# B&R Automation Studio project CleanChemi_SiteManagementSystem (part 9)

```iecst
		// AS Block 125 - ROSTER5_ENABLE
		MasterConfig_LR[IdxSkids_LR].action_enable[124].cyclic := FALSE;// Read data cyclic
		MasterConfig_LR[IdxSkids_LR].action_param[124].p_pv:= ADR(gCMD_LR[IdxSkids_LR].Write_ENABLE_ROSTER5.wENABLE_ROSTER5);// Store data in this variable
		MasterConfig_LR[IdxSkids_LR].action_param[124].quantity := 1;// Number of items to read
		MasterConfig_LR[IdxSkids_LR].action_param[124].unit := 1;// Unit address - ignore if not specified
		MasterConfig_LR[IdxSkids_LR].action_param[124].start_addr := 4560;// Read from this modbus address
		MasterConfig_LR[IdxSkids_LR].action_param[124].timer := 2;// Refresh timer for this item
		MasterConfig_LR[IdxSkids_LR].action_param[124].type := 6;// Function code for this item (2 := read discrete inputs)

		// AS Block 126 - ROSTER6_ENABLE
		MasterConfig_LR[IdxSkids_LR].action_enable[125].cyclic := FALSE;// Read data cyclic
		MasterConfig_LR[IdxSkids_LR].action_param[125].p_pv:= ADR(gCMD_LR[IdxSkids_LR].Write_ENABLE_ROSTER6.wENABLE_ROSTER6);// Store data in this variable
		MasterConfig_LR[IdxSkids_LR].action_param[125].quantity := 1;// Number of items to read
		MasterConfig_LR[IdxSkids_LR].action_param[125].unit := 1;// Unit address - ignore if not specified
		MasterConfig_LR[IdxSkids_LR].action_param[125].start_addr := 4660;// Read from this modbus address
		MasterConfig_LR[IdxSkids_LR].action_param[125].timer := 2;// Refresh timer for this item
		MasterConfig_LR[IdxSkids_LR].action_param[125].type := 6;// Function code for this item (2 := read discrete inputs)

		// AS Block 127 - ROSTER7_ENABLE
		MasterConfig_LR[IdxSkids_LR].action_enable[126].cyclic := FALSE;// Read data cyclic
		MasterConfig_LR[IdxSkids_LR].action_param[126].p_pv:= ADR(gCMD_LR[IdxSkids_LR].Write_ENABLE_ROSTER7.wENABLE_ROSTER7);// Store data in this variable
		MasterConfig_LR[IdxSkids_LR].action_param[126].quantity := 1;// Number of items to read
		MasterConfig_LR[IdxSkids_LR].action_param[126].unit := 1;// Unit address - ignore if not specified
		MasterConfig_LR[IdxSkids_LR].action_param[126].start_addr := 4760;// Read from this modbus address
		MasterConfig_LR[IdxSkids_LR].action_param[126].timer := 2;// Refresh timer for this item
		MasterConfig_LR[IdxSkids_LR].action_param[126].type := 6;// Function code for this item (2 := read discrete inputs)

		// AS Block 128 - ROSTER8_ENABLE
		MasterConfig_LR[IdxSkids_LR].action_enable[127].cyclic := FALSE;// Read data cyclic
		MasterConfig_LR[IdxSkids_LR].action_param[127].p_pv:= ADR(gCMD_LR[IdxSkids_LR].Write_ENABLE_ROSTER8.wENABLE_ROSTER8);// Store data in this variable
		MasterConfig_LR[IdxSkids_LR].action_param[127].quantity := 1;// Number of items to read
		MasterConfig_LR[IdxSkids_LR].action_param[127].unit := 1;// Unit address - ignore if not specified
		MasterConfig_LR[IdxSkids_LR].action_param[127].start_addr := 4860;// Read from this modbus address
		MasterConfig_LR[IdxSkids_LR].action_param[127].timer := 2;// Refresh timer for this item
		MasterConfig_LR[IdxSkids_LR].action_param[127].type := 6;// Function code for this item (2 := read discrete inputs)

		// AS Block 129 - AC_ALARM_ENABLE
		MasterConfig_LR[IdxSkids_LR].action_enable[128].cyclic := FALSE;// Read data cyclic
		MasterConfig_LR[IdxSkids_LR].action_param[128].p_pv:= ADR(gCMD_LR[IdxSkids_LR].Write_AC_ALARM_ENABLE.wAC_ALARM_ENABLE);// Store data in this variable
		MasterConfig_LR[IdxSkids_LR].action_param[128].quantity := 1;// Number of items to read
		MasterConfig_LR[IdxSkids_LR].action_param[128].unit := 1;// Unit address - ignore if not specified
		MasterConfig_LR[IdxSkids_LR].action_param[128].start_addr := gSkid_LR[IdxSkids_LR].AlarmConfig.wAC_ALARM_ENABLE_ADDR;// Read from this modbus address
		MasterConfig_LR[IdxSkids_LR].action_param[128].timer := 2;// Refresh timer for this item
		MasterConfig_LR[IdxSkids_LR].action_param[128].type := 6;// Function code for this item (2 := read discrete inputs)

		// AS Block 130 - AC_TXT_ENABLE
		MasterConfig_LR[IdxSkids_LR].action_enable[129].cyclic := FALSE;// Read data cyclic
		MasterConfig_LR[IdxSkids_LR].action_param[129].p_pv:= ADR(gCMD_LR[IdxSkids_LR].Write_AC_TXT_ENABLE.wAC_TXT_ENABLE);// Store data in this variable
		MasterConfig_LR[IdxSkids_LR].action_param[129].quantity := 1;// Number of items to read
		MasterConfig_LR[IdxSkids_LR].action_param[129].unit := 1;// Unit address - ignore if not specified
		MasterConfig_LR[IdxSkids_LR].action_param[129].start_addr := gSkid_LR[IdxSkids_LR].AlarmConfig.wAC_TXT_ENABLE_ADDR;// Read from this modbus address
		MasterConfig_LR[IdxSkids_LR].action_param[129].timer := 2;// Refresh timer for this item
		MasterConfig_LR[IdxSkids_LR].action_param[129].type := 6;// Function code for this item (2 := read discrete inputs)

		// AS Block 131 - AC_ACTION
		MasterConfig_LR[IdxSkids_LR].action_enable[130].cyclic := FALSE;// Read data cyclic
		MasterConfig_LR[IdxSkids_LR].action_param[130].p_pv:= ADR(gCMD_LR[IdxSkids_LR].Write_AC_ACTION.wAC_ACTION);// Store data in this variable
		MasterConfig_LR[IdxSkids_LR].action_param[130].quantity := 1;// Number of items to read
		MasterConfig_LR[IdxSkids_LR].action_param[130].unit := 1;// Unit address - ignore if not specified
		MasterConfig_LR[IdxSkids_LR].action_param[130].start_addr := gSkid_LR[IdxSkids_LR].AlarmConfig.wAC_ACTION_ADDR;// Read from this modbus address
		MasterConfig_LR[IdxSkids_LR].action_param[130].timer := 2;// Refresh timer for this item
		MasterConfig_LR[IdxSkids_LR].action_param[130].type := 6;// Function code for this item (2 := read discrete inputs)

		// AS Block 132 - AC_DELAY
		MasterConfig_LR[IdxSkids_LR].action_enable[131].cyclic := FALSE;// Read data cyclic
		MasterConfig_LR[IdxSkids_LR].action_param[131].p_pv:= ADR(gCMD_LR[IdxSkids_LR].Write_AC_DELAY.wAC_DELAY);// Store data in this variable
		MasterConfig_LR[IdxSkids_LR].action_param[131].quantity := 1;// Number of items to read
		MasterConfig_LR[IdxSkids_LR].action_param[131].unit := 1;// Unit address - ignore if not specified
		MasterConfig_LR[IdxSkids_LR].action_param[131].start_addr := gSkid_LR[IdxSkids_LR].AlarmConfig.wAC_DELAY_ADDR;// Read from this modbus address
		MasterConfig_LR[IdxSkids_LR].action_param[131].timer := 2;// Refresh timer for this item
		MasterConfig_LR[IdxSkids_LR].action_param[131].type := 6;// Function code for this item (2 := read discrete inputs)

		// AS Block 133 - AC_OFFSET
		MasterConfig_LR[IdxSkids_LR].action_enable[132].cyclic := FALSE;// Read data cyclic
		MasterConfig_LR[IdxSkids_LR].action_param[132].p_pv:= ADR(gCMD_LR[IdxSkids_LR].Write_AC_OFFSET.wAC_OFFSET);// Store data in this variable
		MasterConfig_LR[IdxSkids_LR].action_param[132].quantity := 1;// Number of items to read
		MasterConfig_LR[IdxSkids_LR].action_param[132].unit := 1;// Unit address - ignore if not specified
		MasterConfig_LR[IdxSkids_LR].action_param[132].start_addr := 31000;// Read from this modbus address
		MasterConfig_LR[IdxSkids_LR].action_param[132].timer := 2;// Refresh timer for this item
		MasterConfig_LR[IdxSkids_LR].action_param[132].type := 6;// Function code for this item (2 := read discrete inputs)

		// AS Block 134 - AC_THRESHOLD
		MasterConfig_LR[IdxSkids_LR].action_enable[133].cyclic := FALSE;// Read data cyclic
		MasterConfig_LR[IdxSkids_LR].action_param[133].p_pv:= ADR(gCMD_LR[IdxSkids_LR].Write_AC_THRESHOLD.wAC_THRESHOLD_SWAPPED);// Store data in this variable
		MasterConfig_LR[IdxSkids_LR].action_param[133].quantity := 2;// Number of items to read
		MasterConfig_LR[IdxSkids_LR].action_param[133].unit := 1;// Unit address - ignore if not specified
		MasterConfig_LR[IdxSkids_LR].action_param[133].start_addr := gSkid_LR[IdxSkids_LR].AlarmConfig.wAC_THRESHOLD_ADDR;// Read from this modbus address
		MasterConfig_LR[IdxSkids_LR].action_param[133].timer := 2;// Refresh timer for this item
		MasterConfig_LR[IdxSkids_LR].action_param[133].type := 16;// Function code for this item (2 := read discrete inputs)

		// --------------------------------------------------------------------
		// FOR Modbus Read/Write
		// --------------------------------------------------------------------

		ModbusTcpMaster_LR[IdxSkids_LR].enable := 1;// Start master
		ModbusTcpMaster_LR[IdxSkids_LR].device:= ADR(interface); // Ethernet device string
		ModbusTcpMaster_LR[IdxSkids_LR].p_cfg := ADR(MasterConfig_LR[IdxSkids_LR]); // Pointer to configuration
		ModbusTcpMaster_LR[IdxSkids_LR].p_log := ADR(logger[0,IdxSkids_LR]);// Pointer to logger string array. The logger information will show communication details. Enable for debugging, disable for production to save system resources.
		ModbusTcpMaster_LR[IdxSkids_LR].port:= 510;
		ModbusTcpMaster_LR[IdxSkids_LR].slave_ip_addr := SLAVE_IP_ADDRESSES_LR[IdxSkids_LR]; // Transfer slave device IP address

	END_FOR;

	StartStop := 1;
END_PROGRAM

PROGRAM _CYCLIC
// --------------------------------------------------------------------
// Cyclic FUNCTION call
// --------------------------------------------------------------------
	IF(StartStop) THEN

		FOR IdxSkids_LR := 0 TO MAX_SKIDS_LR DO

			Modbus_CMD_action;
			Modbus_Status_action;
			Alarms_action;

		END_FOR;

	END_IF

END_PROGRAM

PROGRAM _EXIT

	FOR IdxSkids_LR := 0 TO MAX_SKIDS_LR DO
		ModbusTcpMaster_LR[IdxSkids_LR](enable := FALSE);
	END_FOR;

END_PROGRAM
```

#### Status.st
```iecst
ACTION Modbus_Status_action:

	ModbusTcpMaster_LR[IdxSkids_LR]();

	// Heartbeat Connection Monitor
	IF gSkid_LR[IdxSkids_LR].Pmax_General_Variables.HEARTBEAT = gSkid_LR[IdxSkids_LR].Heartbeat.PREVIOUS_HEARTBEAT THEN
		gSkid_LR[IdxSkids_LR].Heartbeat.UNCHANGED_TIMER(IN := TRUE, PT := T#200s);  // Start the timer if value is unchanged for 120 seconds
	ELSE
		gSkid_LR[IdxSkids_LR].Heartbeat.UNCHANGED_TIMER(IN := FALSE);  // Reset the timer if value changes
	END_IF;

	// If the timer reaches 30 seconds, set the systemOffline bit
	IF gSkid_LR[IdxSkids_LR].Heartbeat.UNCHANGED_TIMER.Q THEN
		gSkid_LR[IdxSkids_LR].Heartbeat.SYSTEM_OFFLINE := TRUE;  // System is offline
	ELSE
		gSkid_LR[IdxSkids_LR].Heartbeat.SYSTEM_OFFLINE := FALSE;  // System is still online
	END_IF;

	gSkid_LR[IdxSkids_LR].Heartbeat.MODBUS_RESET(CLK := gSkid_LR[IdxSkids_LR].Heartbeat.SYSTEM_OFFLINE);

	//Reset Modbus buffer on connection timeout
	IF gSkid_LR[IdxSkids_LR].Heartbeat.MODBUS_RESET.Q THEN
		UNIT_ID_Temp := gModbus_LR[IdxSkids_LR].Modbus_PeroxyMAX.Block1_Int[0];
		UNIT_ID_DOSE_Temp := gModbus_LR[IdxSkids_LR].Modbus_Dosing.Block6_Int[0];
		brsmemset(ADR(gModbus_LR[IdxSkids_LR]),0,SIZEOF(gModbus_LR[IdxSkids_LR]));
		gModbus_LR[IdxSkids_LR].Modbus_PeroxyMAX.Block1_Int[0] := UNIT_ID_Temp;
		gModbus_LR[IdxSkids_LR].Modbus_Dosing.Block6_Int[0] := UNIT_ID_DOSE_Temp;
	END_IF;

	// Update previous value for the next cycle
	gSkid_LR[IdxSkids_LR].Heartbeat.PREVIOUS_HEARTBEAT := gSkid_LR[IdxSkids_LR].Pmax_General_Variables.HEARTBEAT;

	// --------------------------------------------------------------------
	// Reset last error information
	// --------------------------------------------------------------------
	IF(reset_error) THEN
		brsmemset(ADR(ModbusTcpMaster_LR[IdxSkids_LR].last_error), 0, 2);
		reset_error := 0;
	END_IF

	// --------------------------------------------------------------------
	// Final Variable Mapping AND Data Conversion - READ
	// --------------------------------------------------------------------

	// AS Block 1 - 6000 DOSING INT
	gSkid_LR[IdxSkids_LR].Pmax_General_Variables.UNIT_ID := gModbus_LR[IdxSkids_LR].Modbus_PeroxyMAX.Block1_Int[0];
	gSkid_LR[IdxSkids_LR].Pmax_General_Variables.USER_ID := gModbus_LR[IdxSkids_LR].Modbus_PeroxyMAX.Block1_Int[2];
	gSkid_LR[IdxSkids_LR].Pmax_General_Variables.USER_ACCESS := gModbus_LR[IdxSkids_LR].Modbus_PeroxyMAX.Block1_Int[4];
	gSkid_LR[IdxSkids_LR].Pmax_General_Variables.PMAX_HOA := gModbus_LR[IdxSkids_LR].Modbus_PeroxyMAX.Block1_Int[6];
	gSkid_LR[IdxSkids_LR].Pmax_General_Variables.PMAX_STATUS := gModbus_LR[IdxSkids_LR].Modbus_PeroxyMAX.Block1_Int[8];
	gSkid_LR[IdxSkids_LR].Pmax_General_Variables.SCREEN_LOCK := INT_TO_BOOL(gModbus_LR[IdxSkids_LR].Modbus_PeroxyMAX.Block1_Int[10]);
	gSkid_LR[IdxSkids_LR].Pmax_General_Variables.HEARTBEAT := gModbus_LR[IdxSkids_LR].Modbus_PeroxyMAX.Block1_Int[12];
	gSkid_LR[IdxSkids_LR].Sensor_Variables.WASTE_LVL := INT_TO_BOOL(gModbus_LR[IdxSkids_LR].Modbus_PeroxyMAX.Block1_Int[14]);

	gSkid_LR[IdxSkids_LR].Pmax_Pump_101.P101_XS := gModbus_LR[IdxSkids_LR].Modbus_PeroxyMAX.Block1_Int[20];
	gSkid_LR[IdxSkids_LR].Sensor_Variables.XV101 := gModbus_LR[IdxSkids_LR].Modbus_PeroxyMAX.Block1_Int[22];
	gSkid_LR[IdxSkids_LR].Sensor_Variables.XV101_ENABLE := gModbus_LR[IdxSkids_LR].Modbus_PeroxyMAX.Block1_Int[24];
	gSkid_LR[IdxSkids_LR].Pmax_Pump_101.P101_AUTOCAL := gModbus_LR[IdxSkids_LR].Modbus_PeroxyMAX.Block1_Int[26];

	gSkid_LR[IdxSkids_LR].Pmax_Pump_102.P102_XS := gModbus_LR[IdxSkids_LR].Modbus_PeroxyMAX.Block1_Int[32];
	gSkid_LR[IdxSkids_LR].Pmax_Pump_102.P102_WARN := gModbus_LR[IdxSkids_LR].Modbus_PeroxyMAX.Block1_Int[34];
	gSkid_LR[IdxSkids_LR].Pmax_Pump_102.P102_ALARM := gModbus_LR[IdxSkids_LR].Modbus_PeroxyMAX.Block1_Int[36];
	gSkid_LR[IdxSkids_LR].Sensor_Variables.XV102 := gModbus_LR[IdxSkids_LR].Modbus_PeroxyMAX.Block1_Int[38];
	gSkid_LR[IdxSkids_LR].Pmax_Pump_102.P102_AUTOCAL := gModbus_LR[IdxSkids_LR].Modbus_PeroxyMAX.Block1_Int[40];
	gSkid_LR[IdxSkids_LR].Pmax_Pump_102.P102_AUTOADAPT := gModbus_LR[IdxSkids_LR].Modbus_PeroxyMAX.Block1_Int[42];
	gSkid_LR[IdxSkids_LR].Pmax_Pump_102.XV102_ENABLE := gModbus_LR[IdxSkids_LR].Modbus_PeroxyMAX.Block1_Int[44];

	gSkid_LR[IdxSkids_LR].Pmax_Pump_103.P103_XS := gModbus_LR[IdxSkids_LR].Modbus_PeroxyMAX.Block1_Int[48];
	gSkid_LR[IdxSkids_LR].Pmax_Pump_103.P103_WARN := gModbus_LR[IdxSkids_LR].Modbus_PeroxyMAX.Block1_Int[50];
	gSkid_LR[IdxSkids_LR].Pmax_Pump_103.P103_ALARM := gModbus_LR[IdxSkids_LR].Modbus_PeroxyMAX.Block1_Int[52];
	gSkid_LR[IdxSkids_LR].Sensor_Variables.XV103 := gModbus_LR[IdxSkids_LR].Modbus_PeroxyMAX.Block1_Int[54];
	gSkid_LR[IdxSkids_LR].Pmax_Pump_103.P103_AUTOCAL := gModbus_LR[IdxSkids_LR].Modbus_PeroxyMAX.Block1_Int[56];
	gSkid_LR[IdxSkids_LR].Pmax_Pump_103.P103_AUTOADAPT := gModbus_LR[IdxSkids_LR].Modbus_PeroxyMAX.Block1_Int[58];

	gSkid_LR[IdxSkids_LR].Pmax_Pump_104.P104_XS := gModbus_LR[IdxSkids_LR].Modbus_PeroxyMAX.Block1_Int[64];
	gSkid_LR[IdxSkids_LR].Pmax_Pump_104.P104_WARN := gModbus_LR[IdxSkids_LR].Modbus_PeroxyMAX.Block1_Int[66];
	gSkid_LR[IdxSkids_LR].Pmax_Pump_104.P104_ALARM := gModbus_LR[IdxSkids_LR].Modbus_PeroxyMAX.Block1_Int[68];
	gSkid_LR[IdxSkids_LR].Sensor_Variables.XV104 := gModbus_LR[IdxSkids_LR].Modbus_PeroxyMAX.Block1_Int[70];
	gSkid_LR[IdxSkids_LR].Pmax_Pump_104.P104_AUTOCAL := gModbus_LR[IdxSkids_LR].Modbus_PeroxyMAX.Block1_Int[72];
	gSkid_LR[IdxSkids_LR].Pmax_Pump_104.P104_AUTOCAL_PV := gModbus_LR[IdxSkids_LR].Modbus_PeroxyMAX.Block1_Int[74];
	gSkid_LR[IdxSkids_LR].Pmax_Pump_104.P104_AUTOADAPT := gModbus_LR[IdxSkids_LR].Modbus_PeroxyMAX.Block1_Int[76];
	gSkid_LR[IdxSkids_LR].Pmax_Pump_104.XV104_ENABLE := gModbus_LR[IdxSkids_LR].Modbus_PeroxyMAX.Block1_Int[78];

	gSkid_LR[IdxSkids_LR].AlarmConfig.AC_ENABLE := gModbus_LR[IdxSkids_LR].Modbus_PeroxyMAX.Block1_Int[118];
	gSkid_LR[IdxSkids_LR].AlarmConfig.AC_ACTION := gModbus_LR[IdxSkids_LR].Modbus_PeroxyMAX.Block1_Int[120];
	gSkid_LR[IdxSkids_LR].AlarmConfig.AC_DELAY := gModbus_LR[IdxSkids_LR].Modbus_PeroxyMAX.Block1_Int[122];
	gSkid_LR[IdxSkids_LR].AlarmConfig.AC_OFFSET := gModbus_LR[IdxSkids_LR].Modbus_PeroxyMAX.Block1_Int[124];

	// AS Block 2 - 6000 DOSING INT - ROSTER
	gSkid_LR[IdxSkids_LR].RosterContact.Contact1_ENABLE := INT_TO_BOOL(gModbus_LR[IdxSkids_LR].Modbus_PeroxyMAX.Block2_Int[0]);
	IDEC_String(ADR(gSkid_LR[IdxSkids_LR].RosterContact.Phone_Read1),ADR(gModbus_LR[IdxSkids_LR].Modbus_PeroxyMAX.Block2_Int[4]),SIZEOF(gSkid_LR[IdxSkids_LR].RosterContact.Phone_Read1),19);

	gSkid_LR[IdxSkids_LR].RosterContact.Contact2_ENABLE := INT_TO_BOOL(gModbus_LR[IdxSkids_LR].Modbus_PeroxyMAX.Block2_Int[24]);
	IDEC_String(ADR(gSkid_LR[IdxSkids_LR].RosterContact.Phone_Read2),ADR(gModbus_LR[IdxSkids_LR].Modbus_PeroxyMAX.Block2_Int[28]),SIZEOF(gSkid_LR[IdxSkids_LR].RosterContact.Phone_Read2),19);

	gSkid_LR[IdxSkids_LR].RosterContact.Contact3_ENABLE := INT_TO_BOOL(gModbus_LR[IdxSkids_LR].Modbus_PeroxyMAX.Block2_Int[48]);
	IDEC_String(ADR(gSkid_LR[IdxSkids_LR].RosterContact.Phone_Read3),ADR(gModbus_LR[IdxSkids_LR].Modbus_PeroxyMAX.Block2_Int[52]),SIZEOF(gSkid_LR[IdxSkids_LR].RosterContact.Phone_Read3),19);

	gSkid_LR[IdxSkids_LR].RosterContact.Contact4_ENABLE := INT_TO_BOOL(gModbus_LR[IdxSkids_LR].Modbus_PeroxyMAX.Block2_Int[72]);
	IDEC_String(ADR(gSkid_LR[IdxSkids_LR].RosterContact.Phone_Read4),ADR(gModbus_LR[IdxSkids_LR].Modbus_PeroxyMAX.Block2_Int[76]),SIZEOF(gSkid_LR[IdxSkids_LR].RosterContact.Phone_Read4),19);

	gSkid_LR[IdxSkids_LR].RosterContact.Contact5_ENABLE := INT_TO_BOOL(gModbus_LR[IdxSkids_LR].Modbus_PeroxyMAX.Block2_Int[96]);
	IDEC_String(ADR(gSkid_LR[IdxSkids_LR].RosterContact.Phone_Read5),ADR(gModbus_LR[IdxSkids_LR].Modbus_PeroxyMAX.Block2_Int[100]),SIZEOF(gSkid_LR[IdxSkids_LR].RosterContact.Phone_Read5),19);

	gSkid_LR[IdxSkids_LR].RosterContact.Contact6_ENABLE := INT_TO_BOOL(gModbus_LR[IdxSkids_LR].Modbus_PeroxyMAX.Block2_Int[120]);
	IDEC_String(ADR(gSkid_LR[IdxSkids_LR].RosterContact.Phone_Read6),ADR(gModbus_LR[IdxSkids_LR].Modbus_PeroxyMAX.Block2_Int[124]),SIZEOF(gSkid_LR[IdxSkids_LR].RosterContact.Phone_Read6),19);

	gSkid_LR[IdxSkids_LR].RosterContact.Contact7_ENABLE := INT_TO_BOOL(gModbus_LR[IdxSkids_LR].Modbus_PeroxyMAX.Block2_Int[144]);
	IDEC_String(ADR(gSkid_LR[IdxSkids_LR].RosterContact.Phone_Read7),ADR(gModbus_LR[IdxSkids_LR].Modbus_PeroxyMAX.Block2_Int[148]),SIZEOF(gSkid_LR[IdxSkids_LR].RosterContact.Phone_Read7),19);

	gSkid_LR[IdxSkids_LR].RosterContact.Contact8_ENABLE := INT_TO_BOOL(gModbus_LR[IdxSkids_LR].Modbus_PeroxyMAX.Block2_Int[168]);
	IDEC_String(ADR(gSkid_LR[IdxSkids_LR].RosterContact.Phone_Read8),ADR(gModbus_LR[IdxSkids_LR].Modbus_PeroxyMAX.Block2_Int[172]),SIZEOF(gSkid_LR[IdxSkids_LR].RosterContact.Phone_Read8),19);

	// AS Block 3 - 6000 DOSING REAL
	gSkid_LR[IdxSkids_LR].ConversionRatios.EFF_1:= IDEC_REAL_Conv(gModbus_LR[IdxSkids_LR].Modbus_PeroxyMAX.Block3_Real[0]);
	gSkid_LR[IdxSkids_LR].ConversionRatios.EFF_2:= IDEC_REAL_Conv(gModbus_LR[IdxSkids_LR].Modbus_PeroxyMAX.Block3_Real[1]);
	gSkid_LR[IdxSkids_LR].ConversionRatios.NAOH_TO_H2O2:= IDEC_REAL_Conv(gModbus_LR[IdxSkids_LR].Modbus_PeroxyMAX.Block3_Real[2]);
	gSkid_LR[IdxSkids_LR].ConversionRatios.TRI_TO_H2O2:= IDEC_REAL_Conv(gModbus_LR[IdxSkids_LR].Modbus_PeroxyMAX.Block3_Real[3]);
	gSkid_LR[IdxSkids_LR].ConversionRatios.NAOH_TO_TRI:= IDEC_REAL_Conv(gModbus_LR[IdxSkids_LR].Modbus_PeroxyMAX.Block3_Real[4]);

	gSkid_LR[IdxSkids_LR].Pmax_General_Variables.PMAX_CONC:= IDEC_REAL_Conv(gModbus_LR[IdxSkids_LR].Modbus_PeroxyMAX.Block3_Real[8]);
	gSkid_LR[IdxSkids_LR].Pmax_General_Variables.PMAX_RATE:= IDEC_REAL_Conv(gModbus_LR[IdxSkids_LR].Modbus_PeroxyMAX.Block3_Real[9]);
	gSkid_LR[IdxSkids_LR].Pmax_General_Variables.PMAX_PV:= IDEC_REAL_Conv(gModbus_LR[IdxSkids_LR].Modbus_PeroxyMAX.Block3_Real[10]);
	gSkid_LR[IdxSkids_LR].Pmax_General_Variables.NAOH_CONC:= IDEC_REAL_Conv(gModbus_LR[IdxSkids_LR].Modbus_PeroxyMAX.Block3_Real[11]);
	gSkid_LR[IdxSkids_LR].Pmax_General_Variables.NAOH_CONC_OD:= IDEC_REAL_Conv(gModbus_LR[IdxSkids_LR].Modbus_PeroxyMAX.Block3_Real[12]);
	gSkid_LR[IdxSkids_LR].Pmax_General_Variables.HP_CONC:= IDEC_REAL_Conv(gModbus_LR[IdxSkids_LR].Modbus_PeroxyMAX.Block3_Real[13]);
	gSkid_LR[IdxSkids_LR].Pmax_General_Variables.HP_CONC_OD:= IDEC_REAL_Conv(gModbus_LR[IdxSkids_LR].Modbus_PeroxyMAX.Block3_Real[14]);

	gSkid_LR[IdxSkids_LR].Pmax_Pump_101.P101_SP:= IDEC_REAL_Conv(gModbus_LR[IdxSkids_LR].Modbus_PeroxyMAX.Block3_Real[21]);
	gSkid_LR[IdxSkids_LR].Pmax_Pump_101.P101_PV:= IDEC_REAL_Conv(gModbus_LR[IdxSkids_LR].Modbus_PeroxyMAX.Block3_Real[22]);
	gSkid_LR[IdxSkids_LR].Pmax_Pump_101.P101_OP:= IDEC_REAL_Conv(gModbus_LR[IdxSkids_LR].Modbus_PeroxyMAX.Block3_Real[23]);
	gSkid_LR[IdxSkids_LR].Pmax_Pump_101.P101_FQ:= IDEC_REAL_Conv(gModbus_LR[IdxSkids_LR].Modbus_PeroxyMAX.Block3_Real[24]);
	gSkid_LR[IdxSkids_LR].Pmax_Pump_101.P101_TI:= IDEC_REAL_Conv(gModbus_LR[IdxSkids_LR].Modbus_PeroxyMAX.Block3_Real[25]);
	gSkid_LR[IdxSkids_LR].Pmax_Pump_101.P101_PI:= IDEC_REAL_Conv(gModbus_LR[IdxSkids_LR].Modbus_PeroxyMAX.Block3_Real[26]);
	gSkid_LR[IdxSkids_LR].Pmax_Pump_101.P101_PFI:= IDEC_REAL_Conv(gModbus_LR[IdxSkids_LR].Modbus_PeroxyMAX.Block3_Real[27]);
	gSkid_LR[IdxSkids_LR].Pmax_Pump_101.P101_LS:= IDEC_REAL_Conv(gModbus_LR[IdxSkids_LR].Modbus_PeroxyMAX.Block3_Real[28]);
	gSkid_LR[IdxSkids_LR].Pmax_Pump_101.P101_GAIN:= IDEC_REAL_Conv(gModbus_LR[IdxSkids_LR].Modbus_PeroxyMAX.Block3_Real[29]);
	gSkid_LR[IdxSkids_LR].Pmax_Pump_101.P101_STEPADJ:= IDEC_REAL_Conv(gModbus_LR[IdxSkids_LR].Modbus_PeroxyMAX.Block3_Real[30]);
	gSkid_LR[IdxSkids_LR].Pmax_Pump_101.P101_TOTALADJ:= IDEC_REAL_Conv(gModbus_LR[IdxSkids_LR].Modbus_PeroxyMAX.Block3_Real[31]);

	gSkid_LR[IdxSkids_LR].Pmax_Pump_101B.P101B_OP:= IDEC_REAL_Conv(gModbus_LR[IdxSkids_LR].Modbus_PeroxyMAX.Block3_Real[35]);
	gSkid_LR[IdxSkids_LR].Pmax_Pump_101B.P101B_PFI:= IDEC_REAL_Conv(gModbus_LR[IdxSkids_LR].Modbus_PeroxyMAX.Block3_Real[36]);
	gSkid_LR[IdxSkids_LR].Pmax_Pump_101B.P101B_SP:= IDEC_REAL_Conv(gModbus_LR[IdxSkids_LR].Modbus_PeroxyMAX.Block3_Real[37]);
	gSkid_LR[IdxSkids_LR].Pmax_Pump_101B.P101B_LS:= IDEC_REAL_Conv(gModbus_LR[IdxSkids_LR].Modbus_PeroxyMAX.Block3_Real[38]);

	gSkid_LR[IdxSkids_LR].Pmax_Pump_102.P102_SP:= IDEC_REAL_Conv(gModbus_LR[IdxSkids_LR].Modbus_PeroxyMAX.Block3_Real[45]);
	gSkid_LR[IdxSkids_LR].Pmax_Pump_102.P102_PV:= IDEC_REAL_Conv(gModbus_LR[IdxSkids_LR].Modbus_PeroxyMAX.Block3_Real[46]);
	gSkid_LR[IdxSkids_LR].Pmax_Pump_102.P102_OP:= IDEC_REAL_Conv(gModbus_LR[IdxSkids_LR].Modbus_PeroxyMAX.Block3_Real[47]);
	gSkid_LR[IdxSkids_LR].Pmax_Pump_102.P102_PFI:= IDEC_REAL_Conv(gModbus_LR[IdxSkids_LR].Modbus_PeroxyMAX.Block3_Real[48]);
	gSkid_LR[IdxSkids_LR].Pmax_Pump_102.P102_FQ:= IDEC_REAL_Conv(gModbus_LR[IdxSkids_LR].Modbus_PeroxyMAX.Block3_Real[49]);
	gSkid_LR[IdxSkids_LR].Pmax_Pump_102.P102_PFQ:= IDEC_REAL_Conv(gModbus_LR[IdxSkids_LR].Modbus_PeroxyMAX.Block3_Real[50]);
	gSkid_LR[IdxSkids_LR].Pmax_Pump_102.P102_PPI:= IDEC_REAL_Conv(gModbus_LR[IdxSkids_LR].Modbus_PeroxyMAX.Block3_Real[51]);
	gSkid_LR[IdxSkids_LR].Pmax_Pump_102.P102_TI:= IDEC_REAL_Conv(gModbus_LR[IdxSkids_LR].Modbus_PeroxyMAX.Block3_Real[52]);
	gSkid_LR[IdxSkids_LR].Pmax_Pump_102.P102_PI:= IDEC_REAL_Conv(gModbus_LR[IdxSkids_LR].Modbus_PeroxyMAX.Block3_Real[53]);
	gSkid_LR[IdxSkids_LR].Pmax_Pump_102.P102_LS:= IDEC_REAL_Conv(gModbus_LR[IdxSkids_LR].Modbus_PeroxyMAX.Block3_Real[54]);
	gSkid_LR[IdxSkids_LR].Pmax_Pump_102.P102_GAIN:= IDEC_REAL_Conv(gModbus_LR[IdxSkids_LR].Modbus_PeroxyMAX.Block3_Real[55]);
	gSkid_LR[IdxSkids_LR].Pmax_Pump_102.P102_STEPADJ:= IDEC_REAL_Conv(gModbus_LR[IdxSkids_LR].Modbus_PeroxyMAX.Block3_Real[56]);
	gSkid_LR[IdxSkids_LR].Pmax_Pump_102.P102_TOTALADJ:= IDEC_REAL_Conv(gModbus_LR[IdxSkids_LR].Modbus_PeroxyMAX.Block3_Real[57]);

	gSkid_LR[IdxSkids_LR].Pmax_Pump_103.P103_SP:= IDEC_REAL_Conv(gModbus_LR[IdxSkids_LR].Modbus_PeroxyMAX.Block3_Real[59]);
	gSkid_LR[IdxSkids_LR].Pmax_Pump_103.P103_PV:= IDEC_REAL_Conv(gModbus_LR[IdxSkids_LR].Modbus_PeroxyMAX.Block3_Real[60]);
	gSkid_LR[IdxSkids_LR].Pmax_Pump_103.P103_OP:= IDEC_REAL_Conv(gModbus_LR[IdxSkids_LR].Modbus_PeroxyMAX.Block3_Real[61]);
	gSkid_LR[IdxSkids_LR].Pmax_Pump_103.P103_PFI:= IDEC_REAL_Conv(gModbus_LR[IdxSkids_LR].Modbus_PeroxyMAX.Block3_Real[62]);

	// AS Block 4 - 6000 DOSING REAL
	gSkid_LR[IdxSkids_LR].Pmax_Pump_103.P103_FQ:= IDEC_REAL_Conv(gModbus_LR[IdxSkids_LR].Modbus_PeroxyMAX.Block4_Real[0]);
	gSkid_LR[IdxSkids_LR].Pmax_Pump_103.P103_PFQ:= IDEC_REAL_Conv(gModbus_LR[IdxSkids_LR].Modbus_PeroxyMAX.Block4_Real[1]);
	gSkid_LR[IdxSkids_LR].Pmax_Pump_103.P103_PPI:= IDEC_REAL_Conv(gModbus_LR[IdxSkids_LR].Modbus_PeroxyMAX.Block4_Real[2]);
	gSkid_LR[IdxSkids_LR].Pmax_Pump_103.P103_TI:= IDEC_REAL_Conv(gModbus_LR[IdxSkids_LR].Modbus_PeroxyMAX.Block4_Real[3]);
	gSkid_LR[IdxSkids_LR].Pmax_Pump_103.P103_PI:= IDEC_REAL_Conv(gModbus_LR[IdxSkids_LR].Modbus_PeroxyMAX.Block4_Real[4]);
	gSkid_LR[IdxSkids_LR].Pmax_Pump_103.P103_LS:= IDEC_REAL_Conv(gModbus_LR[IdxSkids_LR].Modbus_PeroxyMAX.Block4_Real[5]);
	gSkid_LR[IdxSkids_LR].Pmax_Pump_103.P103_GAIN:= IDEC_REAL_Conv(gModbus_LR[IdxSkids_LR].Modbus_PeroxyMAX.Block4_Real[6]);
	gSkid_LR[IdxSkids_LR].Pmax_Pump_103.P103_STEPADJ:= IDEC_REAL_Conv(gModbus_LR[IdxSkids_LR].Modbus_PeroxyMAX.Block4_Real[7]);
	gSkid_LR[IdxSkids_LR].Pmax_Pump_103.P103_TOTALADJ:= IDEC_REAL_Conv(gModbus_LR[IdxSkids_LR].Modbus_PeroxyMAX.Block4_Real[8]);

	gSkid_LR[IdxSkids_LR].Pmax_Pump_104.P104_SP:= IDEC_REAL_Conv(gModbus_LR[IdxSkids_LR].Modbus_PeroxyMAX.Block4_Real[10]);
	gSkid_LR[IdxSkids_LR].Pmax_Pump_104.P104_PV:= IDEC_REAL_Conv(gModbus_LR[IdxSkids_LR].Modbus_PeroxyMAX.Block4_Real[11]);
	gSkid_LR[IdxSkids_LR].Pmax_Pump_104.P104_OP:= IDEC_REAL_Conv(gModbus_LR[IdxSkids_LR].Modbus_PeroxyMAX.Block4_Real[12]);
	gSkid_LR[IdxSkids_LR].Pmax_Pump_104.P104_PFI:= IDEC_REAL_Conv(gModbus_LR[IdxSkids_LR].Modbus_PeroxyMAX.Block4_Real[13]);
	gSkid_LR[IdxSkids_LR].Pmax_Pump_104.P104_FQ:= IDEC_REAL_Conv(gModbus_LR[IdxSkids_LR].Modbus_PeroxyMAX.Block4_Real[14]);
	gSkid_LR[IdxSkids_LR].Pmax_Pump_104.P104_PFQ:= IDEC_REAL_Conv(gModbus_LR[IdxSkids_LR].Modbus_PeroxyMAX.Block4_Real[15]);
	gSkid_LR[IdxSkids_LR].Pmax_Pump_104.P104_PPI:= IDEC_REAL_Conv(gModbus_LR[IdxSkids_LR].Modbus_PeroxyMAX.Block4_Real[16]);
	gSkid_LR[IdxSkids_LR].Pmax_Pump_104.P104_PI:= IDEC_REAL_Conv(gModbus_LR[IdxSkids_LR].Modbus_PeroxyMAX.Block4_Real[18]);
	gSkid_LR[IdxSkids_LR].Pmax_Pump_104.P104_LS:= IDEC_REAL_Conv(gModbus_LR[IdxSkids_LR].Modbus_PeroxyMAX.Block4_Real[19]);
	gSkid_LR[IdxSkids_LR].Pmax_Pump_104.P104_GAIN:= IDEC_REAL_Conv(gModbus_LR[IdxSkids_LR].Modbus_PeroxyMAX.Block4_Real[20]);
	gSkid_LR[IdxSkids_LR].Pmax_Pump_104.P104_STEPADJ:= IDEC_REAL_Conv(gModbus_LR[IdxSkids_LR].Modbus_PeroxyMAX.Block4_Real[21]);
	gSkid_LR[IdxSkids_LR].Pmax_Pump_104.P104_TOTALADJ:= IDEC_REAL_Conv(gModbus_LR[IdxSkids_LR].Modbus_PeroxyMAX.Block4_Real[22]);

	gSkid_LR[IdxSkids_LR].Sensor_Variables.CD101:= IDEC_REAL_Conv(gModbus_LR[IdxSkids_LR].Modbus_PeroxyMAX.Block4_Real[24]);
	gSkid_LR[IdxSkids_LR].Sensor_Variables.CD101_SP:= IDEC_REAL_Conv(gModbus_LR[IdxSkids_LR].Modbus_PeroxyMAX.Block4_Real[25]);
	gSkid_LR[IdxSkids_LR].Sensor_Variables.CD102:= IDEC_REAL_Conv(gModbus_LR[IdxSkids_LR].Modbus_PeroxyMAX.Block4_Real[26]);
	gSkid_LR[IdxSkids_LR].Sensor_Variables.CD102_SP:= IDEC_REAL_Conv(gModbus_LR[IdxSkids_LR].Modbus_PeroxyMAX.Block4_Real[27]);
	gSkid_LR[IdxSkids_LR].Sensor_Variables.CD103:= IDEC_REAL_Conv(gModbus_LR[IdxSkids_LR].Modbus_PeroxyMAX.Block4_Real[28]);
	gSkid_LR[IdxSkids_LR].Sensor_Variables.CD103_SP:= IDEC_REAL_Conv(gModbus_LR[IdxSkids_LR].Modbus_PeroxyMAX.Block4_Real[29]);

	gSkid_LR[IdxSkids_LR].Sensor_Variables.CD101_TI:= IDEC_REAL_Conv(gModbus_LR[IdxSkids_LR].Modbus_PeroxyMAX.Block4_Real[36]);
	gSkid_LR[IdxSkids_LR].Sensor_Variables.CD102_TI:= IDEC_REAL_Conv(gModbus_LR[IdxSkids_LR].Modbus_PeroxyMAX.Block4_Real[37]);
	gSkid_LR[IdxSkids_LR].Sensor_Variables.CD103_TI:= IDEC_REAL_Conv(gModbus_LR[IdxSkids_LR].Modbus_PeroxyMAX.Block4_Real[38]);

	gSkid_LR[IdxSkids_LR].AlarmConfig.AC_THRESHOLD :=  IDEC_REAL_Conv(gModbus_LR[IdxSkids_LR].Modbus_PeroxyMAX.Block4_Real[44]);
	gSkid_LR[IdxSkids_LR].Pmax_General_Variables.HMI_REV_A:= IDEC_REAL_Conv(gModbus_LR[IdxSkids_LR].Modbus_PeroxyMAX.Block4_Real[45]);
	gSkid_LR[IdxSkids_LR].Pmax_General_Variables.HMI_REV_B:= IDEC_REAL_Conv(gModbus_LR[IdxSkids_LR].Modbus_PeroxyMAX.Block4_Real[46]);
	gSkid_LR[IdxSkids_LR].Pmax_General_Variables.PLC_REV_A:= IDEC_REAL_Conv(gModbus_LR[IdxSkids_LR].Modbus_PeroxyMAX.Block4_Real[47]);
	gSkid_LR[IdxSkids_LR].Pmax_General_Variables.PLC_REV_B:= IDEC_REAL_Conv(gModbus_LR[IdxSkids_LR].Modbus_PeroxyMAX.Block4_Real[48]);

	gSkid_LR[IdxSkids_LR].BufferTank.BT_PERCENT:= IDEC_REAL_Conv(gModbus_LR[IdxSkids_LR].Modbus_PeroxyMAX.Block4_Real[50]);
	gSkid_LR[IdxSkids_LR].BufferTank.LI200:= IDEC_REAL_Conv(gModbus_LR[IdxSkids_LR].Modbus_PeroxyMAX.Block4_Real[51]);
	gSkid_LR[IdxSkids_LR].BufferTank.LSHH200:= IDEC_REAL_Conv(gModbus_LR[IdxSkids_LR].Modbus_PeroxyMAX.Block4_Real[52]);
	gSkid_LR[IdxSkids_LR].BufferTank.DRAINTIME_SP:= IDEC_REAL_Conv(gModbus_LR[IdxSkids_LR].Modbus_PeroxyMAX.Block4_Real[53]);
	gSkid_LR[IdxSkids_LR].BufferTank.DRAINTIME_PV:= IDEC_REAL_Conv(gModbus_LR[IdxSkids_LR].Modbus_PeroxyMAX.Block4_Real[54]);
	gSkid_LR[IdxSkids_LR].BufferTank.FILLTIME_SP:= IDEC_REAL_Conv(gModbus_LR[IdxSkids_LR].Modbus_PeroxyMAX.Block4_Real[55]);
	gSkid_LR[IdxSkids_LR].BufferTank.FILLTIME_PV:= IDEC_REAL_Conv(gModbus_LR[IdxSkids_LR].Modbus_PeroxyMAX.Block4_Real[56]);

	// AS Block 5 - 6000 DOSING REAL - SPARE
	//:= IDEC_REAL_Conv(gModbus_LR[IdxSkids_LR].Modbus_PeroxyMAX.Block5_Real[0]);

	// AS Block 6 - 7000 DOSING INT
	gSkid_LR[IdxSkids_LR].Pmax_General_Variables.UNIT_ID_DOSE := gModbus_LR[IdxSkids_LR].Modbus_Dosing.Block6_Int[0];

	gSkid_LR[IdxSkids_LR].Dosing_Pump_201.P201_XS := gModbus_LR[IdxSkids_LR].Modbus_Dosing.Block6_Int[6];
	gSkid_LR[IdxSkids_LR].Dosing_Pump_201.P201_HOA := gModbus_LR[IdxSkids_LR].Modbus_Dosing.Block6_Int[8];
	gSkid_LR[IdxSkids_LR].Dosing_Pump_201.P201_CHEM := gModbus_LR[IdxSkids_LR].Modbus_Dosing.Block6_Int[10];
	gSkid_LR[IdxSkids_LR].Dosing_Pump_201.P201_ENABLE := gModbus_LR[IdxSkids_LR].Modbus_Dosing.Block6_Int[12];
	gSkid_LR[IdxSkids_LR].Dosing_Pump_201.P201_ADJ := gModbus_LR[IdxSkids_LR].Modbus_Dosing.Block6_Int[14];
	gSkid_LR[IdxSkids_LR].Dosing_Pump_201.P201_PTYPE := gModbus_LR[IdxSkids_LR].Modbus_Dosing.Block6_Int[16];
	gSkid_LR[IdxSkids_LR].Dosing_Pump_201.P201_WARN := gModbus_LR[IdxSkids_LR].Modbus_Dosing.Block6_Int[18];
	gSkid_LR[IdxSkids_LR].Dosing_Pump_201.P201_ALARM := gModbus_LR[IdxSkids_LR].Modbus_Dosing.Block6_Int[20];
	gSkid_LR[IdxSkids_LR].Sensor_Variables.XV201 := gModbus_LR[IdxSkids_LR].Modbus_Dosing.Block6_Int[22];
	gSkid_LR[IdxSkids_LR].Dosing_Pump_201.P201_AUTOCAL := gModbus_LR[IdxSkids_LR].Modbus_Dosing.Block6_Int[24];
	gSkid_LR[IdxSkids_LR].Dosing_Pump_201.P201_AUTOCAL_PV := gModbus_LR[IdxSkids_LR].Modbus_Dosing.Block6_Int[26];
	gSkid_LR[IdxSkids_LR].Dosing_Pump_201.P201_AUTOADAPT := gModbus_LR[IdxSkids_LR].Modbus_Dosing.Block6_Int[28];

	gSkid_LR[IdxSkids_LR].Dosing_Pump_202.P202_XS := gModbus_LR[IdxSkids_LR].Modbus_Dosing.Block6_Int[32];
	gSkid_LR[IdxSkids_LR].Dosing_Pump_202.P202_HOA := gModbus_LR[IdxSkids_LR].Modbus_Dosing.Block6_Int[34];
	gSkid_LR[IdxSkids_LR].Dosing_Pump_202.P202_CHEM := gModbus_LR[IdxSkids_LR].Modbus_Dosing.Block6_Int[36];
	gSkid_LR[IdxSkids_LR].Dosing_Pump_202.P202_ENABLE := gModbus_LR[IdxSkids_LR].Modbus_Dosing.Block6_Int[38];
	gSkid_LR[IdxSkids_LR].Dosing_Pump_202.P202_ADJ := gModbus_LR[IdxSkids_LR].Modbus_Dosing.Block6_Int[40];
	gSkid_LR[IdxSkids_LR].Dosing_Pump_202.P202_WARN := gModbus_LR[IdxSkids_LR].Modbus_Dosing.Block6_Int[42];
	gSkid_LR[IdxSkids_LR].Dosing_Pump_202.P202_ALARM := gModbus_LR[IdxSkids_LR].Modbus_Dosing.Block6_Int[44];
	gSkid_LR[IdxSkids_LR].Sensor_Variables.XV202 := gModbus_LR[IdxSkids_LR].Modbus_Dosing.Block6_Int[46];
	gSkid_LR[IdxSkids_LR].Dosing_Pump_202.P202_AUTOCAL := gModbus_LR[IdxSkids_LR].Modbus_Dosing.Block6_Int[48];
	gSkid_LR[IdxSkids_LR].Dosing_Pump_202.P202_AUTOCAL_PV := gModbus_LR[IdxSkids_LR].Modbus_Dosing.Block6_Int[50];
	gSkid_LR[IdxSkids_LR].Dosing_Pump_202.P202_AUTOADAPT := gModbus_LR[IdxSkids_LR].Modbus_Dosing.Block6_Int[52];

	gSkid_LR[IdxSkids_LR].Dosing_Pump_203.P203_XS := gModbus_LR[IdxSkids_LR].Modbus_Dosing.Block6_Int[56];
	gSkid_LR[IdxSkids_LR].Dosing_Pump_203.P203_HOA := gModbus_LR[IdxSkids_LR].Modbus_Dosing.Block6_Int[58];
	gSkid_LR[IdxSkids_LR].Dosing_Pump_203.P203_CHEM := gModbus_LR[IdxSkids_LR].Modbus_Dosing.Block6_Int[60];
	gSkid_LR[IdxSkids_LR].Dosing_Pump_203.P203_ENABLE := gModbus_LR[IdxSkids_LR].Modbus_Dosing.Block6_Int[62];
	gSkid_LR[IdxSkids_LR].Dosing_Pump_203.P203_ADJ := gModbus_LR[IdxSkids_LR].Modbus_Dosing.Block6_Int[64];
	gSkid_LR[IdxSkids_LR].Dosing_Pump_203.P203_WARN := gModbus_LR[IdxSkids_LR].Modbus_Dosing.Block6_Int[66];
	gSkid_LR[IdxSkids_LR].Dosing_Pump_203.P203_ALARM := gModbus_LR[IdxSkids_LR].Modbus_Dosing.Block6_Int[68];
	gSkid_LR[IdxSkids_LR].Sensor_Variables.XV203 := gModbus_LR[IdxSkids_LR].Modbus_Dosing.Block6_Int[70];
	gSkid_LR[IdxSkids_LR].Dosing_Pump_203.P203_AUTOCAL := gModbus_LR[IdxSkids_LR].Modbus_Dosing.Block6_Int[72];
	gSkid_LR[IdxSkids_LR].Dosing_Pump_203.P203_AUTOCAL_PV := gModbus_LR[IdxSkids_LR].Modbus_Dosing.Block6_Int[74];
	gSkid_LR[IdxSkids_LR].Dosing_Pump_203.P203_AUTOADAPT := gModbus_LR[IdxSkids_LR].Modbus_Dosing.Block6_Int[76];

	// AS Block 7 - 7000 DOSING INT
	gSkid_LR[IdxSkids_LR].Sensor_Variables.SERNSORS_CONFIG := gModbus_LR[IdxSkids_LR].Modbus_Dosing.Block7_Int[104];

	gSkid_LR[IdxSkids_LR].Sensor_Variables.FI301_MODE := gModbus_LR[IdxSkids_LR].Modbus_Dosing.Block7_Int[118];
	gSkid_LR[IdxSkids_LR].Sensor_Variables.FI302_MODE := gModbus_LR[IdxSkids_LR].Modbus_Dosing.Block7_Int[120];
	gSkid_LR[IdxSkids_LR].Sensor_Variables.FI303_MODE := gModbus_LR[IdxSkids_LR].Modbus_Dosing.Block7_Int[122];
	gSkid_LR[IdxSkids_LR].Sensor_Variables.FI304_MODE := gModbus_LR[IdxSkids_LR].Modbus_Dosing.Block7_Int[124];

	// AS Block 8 - 7000 DOSING REAL
	gSkid_LR[IdxSkids_LR].Dosing_Pump_201.P201_REF_SENSOR := IDEC_REAL_Conv(gModbus_LR[IdxSkids_LR].Modbus_Dosing.Block8_Real[0]);
	gSkid_LR[IdxSkids_LR].Dosing_Pump_201.P201_CONC := IDEC_REAL_Conv(gModbus_LR[IdxSkids_LR].Modbus_Dosing.Block8_Real[1]);
	gSkid_LR[IdxSkids_LR].Dosing_Pump_201.P201_PPM := IDEC_REAL_Conv(gModbus_LR[IdxSkids_LR].Modbus_Dosing.Block8_Real[2]);
	gSkid_LR[IdxSkids_LR].Dosing_Pump_201.P201_APPM := IDEC_REAL_Conv(gModbus_LR[IdxSkids_LR].Modbus_Dosing.Block8_Real[3]);
	gSkid_LR[IdxSkids_LR].Dosing_Pump_201.P201_SP := IDEC_REAL_Conv(gModbus_LR[IdxSkids_LR].Modbus_Dosing.Block8_Real[4]);
	gSkid_LR[IdxSkids_LR].Dosing_Pump_201.P201_PV := IDEC_REAL_Conv(gModbus_LR[IdxSkids_LR].Modbus_Dosing.Block8_Real[5]);
	gSkid_LR[IdxSkids_LR].Dosing_Pump_201.P201_OP := IDEC_REAL_Conv(gModbus_LR[IdxSkids_LR].Modbus_Dosing.Block8_Real[6]);
	gSkid_LR[IdxSkids_LR].Dosing_Pump_201.P201_PFI := IDEC_REAL_Conv(gModbus_LR[IdxSkids_LR].Modbus_Dosing.Block8_Real[7]);
	gSkid_LR[IdxSkids_LR].Dosing_Pump_201.P201_FQ := IDEC_REAL_Conv(gModbus_LR[IdxSkids_LR].Modbus_Dosing.Block8_Real[8]);
	gSkid_LR[IdxSkids_LR].Dosing_Pump_201.P201_PI := IDEC_REAL_Conv(gModbus_LR[IdxSkids_LR].Modbus_Dosing.Block8_Real[9]);
	gSkid_LR[IdxSkids_LR].Dosing_Pump_201.P201_TI := IDEC_REAL_Conv(gModbus_LR[IdxSkids_LR].Modbus_Dosing.Block8_Real[10]);
	gSkid_LR[IdxSkids_LR].Dosing_Pump_201.P201_PFQ := IDEC_REAL_Conv(gModbus_LR[IdxSkids_LR].Modbus_Dosing.Block8_Real[11]);
	gSkid_LR[IdxSkids_LR].Dosing_Pump_201.P201_PPI := IDEC_REAL_Conv(gModbus_LR[IdxSkids_LR].Modbus_Dosing.Block8_Real[12]);
	gSkid_LR[IdxSkids_LR].Dosing_Pump_201.P201_LS := IDEC_REAL_Conv(gModbus_LR[IdxSkids_LR].Modbus_Dosing.Block8_Real[13]);
	gSkid_LR[IdxSkids_LR].Dosing_Pump_201.P201_ASP := IDEC_REAL_Conv(gModbus_LR[IdxSkids_LR].Modbus_Dosing.Block8_Real[14]);
	gSkid_LR[IdxSkids_LR].Dosing_Pump_201.P201_GAIN := IDEC_REAL_Conv(gModbus_LR[IdxSkids_LR].Modbus_Dosing.Block8_Real[15]);
	gSkid_LR[IdxSkids_LR].Dosing_Pump_201.P201_STEPADJ := IDEC_REAL_Conv(gModbus_LR[IdxSkids_LR].Modbus_Dosing.Block8_Real[16]);
	gSkid_LR[IdxSkids_LR].Dosing_Pump_201.P201_TOTALADJ := IDEC_REAL_Conv(gModbus_LR[IdxSkids_LR].Modbus_Dosing.Block8_Real[17]);

	gSkid_LR[IdxSkids_LR].Dosing_Pump_202.P202_REF_SENSOR := IDEC_REAL_Conv(gModbus_LR[IdxSkids_LR].Modbus_Dosing.Block8_Real[19]);
	gSkid_LR[IdxSkids_LR].Dosing_Pump_202.P202_CONC := IDEC_REAL_Conv(gModbus_LR[IdxSkids_LR].Modbus_Dosing.Block8_Real[20]);
	gSkid_LR[IdxSkids_LR].Dosing_Pump_202.P202_PPM := IDEC_REAL_Conv(gModbus_LR[IdxSkids_LR].Modbus_Dosing.Block8_Real[21]);
	gSkid_LR[IdxSkids_LR].Dosing_Pump_202.P202_APPM := IDEC_REAL_Conv(gModbus_LR[IdxSkids_LR].Modbus_Dosing.Block8_Real[22]);
	gSkid_LR[IdxSkids_LR].Dosing_Pump_202.P202_SP := IDEC_REAL_Conv(gModbus_LR[IdxSkids_LR].Modbus_Dosing.Block8_Real[23]);
	gSkid_LR[IdxSkids_LR].Dosing_Pump_202.P202_PV := IDEC_REAL_Conv(gModbus_LR[IdxSkids_LR].Modbus_Dosing.Block8_Real[24]);
	gSkid_LR[IdxSkids_LR].Dosing_Pump_202.P202_OP := IDEC_REAL_Conv(gModbus_LR[IdxSkids_LR].Modbus_Dosing.Block8_Real[25]);
	gSkid_LR[IdxSkids_LR].Dosing_Pump_202.P202_PFI := IDEC_REAL_Conv(gModbus_LR[IdxSkids_LR].Modbus_Dosing.Block8_Real[26]);
	gSkid_LR[IdxSkids_LR].Dosing_Pump_202.P202_FQ := IDEC_REAL_Conv(gModbus_LR[IdxSkids_LR].Modbus_Dosing.Block8_Real[27]);
	gSkid_LR[IdxSkids_LR].Dosing_Pump_202.P202_PI := IDEC_REAL_Conv(gModbus_LR[IdxSkids_LR].Modbus_Dosing.Block8_Real[28]);
	gSkid_LR[IdxSkids_LR].Dosing_Pump_202.P202_TI := IDEC_REAL_Conv(gModbus_LR[IdxSkids_LR].Modbus_Dosing.Block8_Real[29]);
	gSkid_LR[IdxSkids_LR].Dosing_Pump_202.P202_PFQ := IDEC_REAL_Conv(gModbus_LR[IdxSkids_LR].Modbus_Dosing.Block8_Real[30]);
	gSkid_LR[IdxSkids_LR].Dosing_Pump_202.P202_PPI := IDEC_REAL_Conv(gModbus_LR[IdxSkids_LR].Modbus_Dosing.Block8_Real[31]);
	gSkid_LR[IdxSkids_LR].Dosing_Pump_202.P202_LS := IDEC_REAL_Conv(gModbus_LR[IdxSkids_LR].Modbus_Dosing.Block8_Real[32]);
	gSkid_LR[IdxSkids_LR].Dosing_Pump_202.P202_ASP := IDEC_REAL_Conv(gModbus_LR[IdxSkids_LR].Modbus_Dosing.Block8_Real[33]);
	gSkid_LR[IdxSkids_LR].Dosing_Pump_202.P202_GAIN := IDEC_REAL_Conv(gModbus_LR[IdxSkids_LR].Modbus_Dosing.Block8_Real[34]);
	gSkid_LR[IdxSkids_LR].Dosing_Pump_202.P202_STEPADJ := IDEC_REAL_Conv(gModbus_LR[IdxSkids_LR].Modbus_Dosing.Block8_Real[35]);
	gSkid_LR[IdxSkids_LR].Dosing_Pump_202.P202_TOTALADJ := IDEC_REAL_Conv(gModbus_LR[IdxSkids_LR].Modbus_Dosing.Block8_Real[36]);

	gSkid_LR[IdxSkids_LR].Dosing_Pump_203.P203_REF_SENSOR := IDEC_REAL_Conv(gModbus_LR[IdxSkids_LR].Modbus_Dosing.Block8_Real[38]);
	gSkid_LR[IdxSkids_LR].Dosing_Pump_203.P203_CONC := IDEC_REAL_Conv(gModbus_LR[IdxSkids_LR].Modbus_Dosing.Block8_Real[39]);
	gSkid_LR[IdxSkids_LR].Dosing_Pump_203.P203_PPM := IDEC_REAL_Conv(gModbus_LR[IdxSkids_LR].Modbus_Dosing.Block8_Real[40]);
	gSkid_LR[IdxSkids_LR].Dosing_Pump_203.P203_APPM := IDEC_REAL_Conv(gModbus_LR[IdxSkids_LR].Modbus_Dosing.Block8_Real[41]);
	gSkid_LR[IdxSkids_LR].Dosing_Pump_203.P203_SP := IDEC_REAL_Conv(gModbus_LR[IdxSkids_LR].Modbus_Dosing.Block8_Real[42]);
	gSkid_LR[IdxSkids_LR].Dosing_Pump_203.P203_PV := IDEC_REAL_Conv(gModbus_LR[IdxSkids_LR].Modbus_Dosing.Block8_Real[43]);
	gSkid_LR[IdxSkids_LR].Dosing_Pump_203.P203_OP := IDEC_REAL_Conv(gModbus_LR[IdxSkids_LR].Modbus_Dosing.Block8_Real[44]);
	gSkid_LR[IdxSkids_LR].Dosing_Pump_203.P203_PFI := IDEC_REAL_Conv(gModbus_LR[IdxSkids_LR].Modbus_Dosing.Block8_Real[45]);
	gSkid_LR[IdxSkids_LR].Dosing_Pump_203.P203_FQ := IDEC_REAL_Conv(gModbus_LR[IdxSkids_LR].Modbus_Dosing.Block8_Real[46]);
	gSkid_LR[IdxSkids_LR].Dosing_Pump_203.P203_PI := IDEC_REAL_Conv(gModbus_LR[IdxSkids_LR].Modbus_Dosing.Block8_Real[47]);
	gSkid_LR[IdxSkids_LR].Dosing_Pump_203.P203_TI := IDEC_REAL_Conv(gModbus_LR[IdxSkids_LR].Modbus_Dosing.Block8_Real[48]);
	gSkid_LR[IdxSkids_LR].Dosing_Pump_203.P203_PFQ := IDEC_REAL_Conv(gModbus_LR[IdxSkids_LR].Modbus_Dosing.Block8_Real[49]);
	gSkid_LR[IdxSkids_LR].Dosing_Pump_203.P203_PPI := IDEC_REAL_Conv(gModbus_LR[IdxSkids_LR].Modbus_Dosing.Block8_Real[50]);
	gSkid_LR[IdxSkids_LR].Dosing_Pump_203.P203_LS := IDEC_REAL_Conv(gModbus_LR[IdxSkids_LR].Modbus_Dosing.Block8_Real[51]);
	gSkid_LR[IdxSkids_LR].Dosing_Pump_203.P203_ASP := IDEC_REAL_Conv(gModbus_LR[IdxSkids_LR].Modbus_Dosing.Block8_Real[52]);
	gSkid_LR[IdxSkids_LR].Dosing_Pump_203.P203_GAIN := IDEC_REAL_Conv(gModbus_LR[IdxSkids_LR].Modbus_Dosing.Block8_Real[53]);
	gSkid_LR[IdxSkids_LR].Dosing_Pump_203.P203_STEPADJ := IDEC_REAL_Conv(gModbus_LR[IdxSkids_LR].Modbus_Dosing.Block8_Real[54]);
	gSkid_LR[IdxSkids_LR].Dosing_Pump_203.P203_TOTALADJ := IDEC_REAL_Conv(gModbus_LR[IdxSkids_LR].Modbus_Dosing.Block8_Real[55]);

	// AS Block 9 - 7000 DOSING REAL
	//:= IDEC_REAL_Conv(gModbus_LR[IdxSkids_LR].Modbus_Dosing.Block9_Real[0]);

	// AS Block 10 - 7000 DOSING REAL
	gSkid_LR[IdxSkids_LR].Sensor_Variables.SENSOR301 := IDEC_REAL_Conv(gModbus_LR[IdxSkids_LR].Modbus_Dosing.Block10_Real[26]);
	gSkid_LR[IdxSkids_LR].Sensor_Variables.SENSOR302 := IDEC_REAL_Conv(gModbus_LR[IdxSkids_LR].Modbus_Dosing.Block10_Real[27]);
	gSkid_LR[IdxSkids_LR].Sensor_Variables.SENSOR303 := IDEC_REAL_Conv(gModbus_LR[IdxSkids_LR].Modbus_Dosing.Block10_Real[28]);
	gSkid_LR[IdxSkids_LR].Sensor_Variables.SENSOR304 := IDEC_REAL_Conv(gModbus_LR[IdxSkids_LR].Modbus_Dosing.Block10_Real[29]);

	gSkid_LR[IdxSkids_LR].Sensor_Variables.FI301 := IDEC_REAL_Conv(gModbus_LR[IdxSkids_LR].Modbus_Dosing.Block10_Real[34]);
	gSkid_LR[IdxSkids_LR].Sensor_Variables.FI301_QT := IDEC_REAL_Conv(gModbus_LR[IdxSkids_LR].Modbus_Dosing.Block10_Real[35]);
	gSkid_LR[IdxSkids_LR].Sensor_Variables.FI302 := IDEC_REAL_Conv(gModbus_LR[IdxSkids_LR].Modbus_Dosing.Block10_Real[36]);
	gSkid_LR[IdxSkids_LR].Sensor_Variables.FI302_QT := IDEC_REAL_Conv(gModbus_LR[IdxSkids_LR].Modbus_Dosing.Block10_Real[37]);
	gSkid_LR[IdxSkids_LR].Sensor_Variables.FI303 := IDEC_REAL_Conv(gModbus_LR[IdxSkids_LR].Modbus_Dosing.Block10_Real[38]);
	gSkid_LR[IdxSkids_LR].Sensor_Variables.FI303_QT := IDEC_REAL_Conv(gModbus_LR[IdxSkids_LR].Modbus_Dosing.Block10_Real[39]);
	gSkid_LR[IdxSkids_LR].Sensor_Variables.FI304 := IDEC_REAL_Conv(gModbus_LR[IdxSkids_LR].Modbus_Dosing.Block10_Real[40]);
	gSkid_LR[IdxSkids_LR].Sensor_Variables.FI304_QT := IDEC_REAL_Conv(gModbus_LR[IdxSkids_LR].Modbus_Dosing.Block10_Real[41]);

	// AS Block 11 - 7000 DOSING REAL - SPARE
	//:= IDEC_REAL_Conv(gModbus_LR[IdxSkids_LR].Modbus_Dosing.Block11_Real[0]);

	// AS Block 48 - ALARMS
	gSkid_LR[IdxSkids_LR].Alarms.ALARM_AB1 := gModbus_LR[IdxSkids_LR].Modbus_Alarms.Block48_Int[0];
	gSkid_LR[IdxSkids_LR].Alarms.ALARM_AB2 := gModbus_LR[IdxSkids_LR].Modbus_Alarms.Block48_Int[1];
	gSkid_LR[IdxSkids_LR].Alarms.ALARM_AB3 := gModbus_LR[IdxSkids_LR].Modbus_Alarms.Block48_Int[2];
	gSkid_LR[IdxSkids_LR].Alarms.ALARM_AB4 := gModbus_LR[IdxSkids_LR].Modbus_Alarms.Block48_Int[3];
	gSkid_LR[IdxSkids_LR].Alarms.ALARM_AB5 := gModbus_LR[IdxSkids_LR].Modbus_Alarms.Block48_Int[4];
	gSkid_LR[IdxSkids_LR].Alarms.ALARM_AB6 := gModbus_LR[IdxSkids_LR].Modbus_Alarms.Block48_Int[5];
	gSkid_LR[IdxSkids_LR].Alarms.ALARM_AB7 := gModbus_LR[IdxSkids_LR].Modbus_Alarms.Block48_Int[6];
	gSkid_LR[IdxSkids_LR].Alarms.ALARM_AB8 := gModbus_LR[IdxSkids_LR].Modbus_Alarms.Block48_Int[7];
	gSkid_LR[IdxSkids_LR].Alarms.ALARM_AB9 := gModbus_LR[IdxSkids_LR].Modbus_Alarms.Block48_Int[8];
	gSkid_LR[IdxSkids_LR].Alarms.ALARM_AB10 := gModbus_LR[IdxSkids_LR].Modbus_Alarms.Block48_Int[9];
	gSkid_LR[IdxSkids_LR].Alarms.ALARM_AB11 := gModbus_LR[IdxSkids_LR].Modbus_Alarms.Block48_Int[10];

	gSkid_LR[IdxSkids_LR].Alarms.ALARM_AB12 := gModbus_LR[IdxSkids_LR].Modbus_Alarms.Block48_Int[51];
	gSkid_LR[IdxSkids_LR].Alarms.ALARM_AB13 := gModbus_LR[IdxSkids_LR].Modbus_Alarms.Block48_Int[52];
	gSkid_LR[IdxSkids_LR].Alarms.ALARM_AB14 := gModbus_LR[IdxSkids_LR].Modbus_Alarms.Block48_Int[53];
	gSkid_LR[IdxSkids_LR].Alarms.ALARM_AB15 := gModbus_LR[IdxSkids_LR].Modbus_Alarms.Block48_Int[54];
	gSkid_LR[IdxSkids_LR].Alarms.ALARM_AB16 := gModbus_LR[IdxSkids_LR].Modbus_Alarms.Block48_Int[55];
	gSkid_LR[IdxSkids_LR].Alarms.ALARM_AB17 := gModbus_LR[IdxSkids_LR].Modbus_Alarms.Block48_Int[56];
	gSkid_LR[IdxSkids_LR].Alarms.ALARM_AB18 := gModbus_LR[IdxSkids_LR].Modbus_Alarms.Block48_Int[57];
	gSkid_LR[IdxSkids_LR].Alarms.ALARM_AB19 := gModbus_LR[IdxSkids_LR].Modbus_Alarms.Block48_Int[58];

	// AS Block 61 - DOSING PUMP TEXT
	IDEC_String(ADR(gSkid_LR[IdxSkids_LR].Dosing_Pump_201.P201_TEXT),ADR(gModbus_LR[IdxSkids_LR].Modbus_Dosing.Block61_Int[0]),SIZEOF(gSkid_LR[IdxSkids_LR].Dosing_Pump_201.P201_TEXT),27);
	IDEC_String(ADR(gSkid_LR[IdxSkids_LR].Dosing_Pump_202.P202_TEXT),ADR(gModbus_LR[IdxSkids_LR].Modbus_Dosing.Block61_Int[28]),SIZEOF(gSkid_LR[IdxSkids_LR].Dosing_Pump_202.P202_TEXT),27);
	IDEC_String(ADR(gSkid_LR[IdxSkids_LR].Dosing_Pump_203.P203_TEXT),ADR(gModbus_LR[IdxSkids_LR].Modbus_Dosing.Block61_Int[56]),SIZEOF(gSkid_LR[IdxSkids_LR].Dosing_Pump_203.P203_TEXT),27);

END_ACTION
```

### Library Logical/modbusTCP/IDEC_Real (IEC)

#### IDEC_Real.fun - Exported functions and function blocks
```iecst
FUNCTION IDEC_REAL_Conv : REAL
	VAR_INPUT
		REAL_FROM_IDEC : REAL;
	END_VAR
	VAR
		Real_Temp : REAL;
	END_VAR
END_FUNCTION
```

#### IDEC_REAL_Conv.st
```iecst
(* TODO: Add your comment here *)

FUNCTION IDEC_REAL_Conv

	brsmemmove(ADR(Real_Temp) + 2,ADR(REAL_FROM_IDEC),2);
	brsmemmove(ADR(Real_Temp),ADR(REAL_FROM_IDEC)+2,2);

	IDEC_REAL_Conv := Real_Temp;

END_FUNCTION
```

### Library Logical/modbusTCP/IDEC_Strng (IEC)

#### IDEC_Strng.fun
```iecst
{REDUND_ERROR} FUNCTION IDEC_String : BOOL (*TODO: Add your comment here*) (*$GROUP=User,$CAT=User,$GROUPICON=User.png,$CATICON=User.png*)
	VAR_INPUT
		pDest : UDINT;
		pSrc : UDINT;
		SizeDest : UDINT;
		SizeSrc : UDINT;
	END_VAR
	VAR
		j : USINT;
		i : UDINT;
	END_VAR
END_FUNCTION
```

#### IDEC_String.st
```iecst
(* TODO: Add your comment here *)
FUNCTION IDEC_String

	FOR i := 0 TO SizeSrc BY 4 DO
		brsmemcpy(pDest+(j+1),pSrc+i,1);
		brsmemcpy(pDest+j,pSrc+(i+1),1);
		j := j+2;
	END_FOR;

END_FUNCTION
```

### Library Logical/modbusTCP/HA_JSON (IEC)
Depends on: HA_Str, AsBrStr, sys_lib

#### HA_JSON.fun - Exported functions and function blocks
```iecst
{REDUND_ERROR} FUNCTION_BLOCK HA_JSON_PairsToJSON (*FB parses a JSON string into a flat array of Name and Value Pairs*) (*$GROUP=User,$CAT=User,$GROUPICON=User.png,$CATICON=User.png*)
	VAR_INPUT
		Enable : BOOL;
		pBuffer : UDINT; (*Pointer to Buffer*)
		BufferSIZEOF : UDINT; (*Buffer SIZEOF*)
		pPairs : UDINT; (*Pointer to Array defined as HA_JSON_Parse_Pair_typ[0..MAX_JSON_PARSE_PAIR_IDX]*)
	END_VAR
	VAR_OUTPUT
		Done : BOOL;
		Error : BOOL;
	END_VAR
	VAR
		Internal : HA_JSON_PairsToJSON_Internal_typ;
	END_VAR
END_FUNCTION_BLOCK

{REDUND_ERROR} FUNCTION_BLOCK HA_JSON_Parse (*FB parses a JSON string into a flat array of Name and Value Pairs*) (*$GROUP=User,$CAT=User,$GROUPICON=User.png,$CATICON=User.png*)
	VAR_INPUT
		Enable : BOOL;
		pBuffer : UDINT; (*Pointer to Buffer*)
		pPairs : UDINT; (*Pointer to Array defined as HA_JSON_Parse_Pair_typ[0..MAX_JSON_PARSE_PAIR_IDX]*)
	END_VAR
	VAR_OUTPUT
		Done : BOOL;
		Error : BOOL;
	END_VAR
	VAR
		Internal : HA_JSON_Parse_Internal_typ;
	END_VAR
END_FUNCTION_BLOCK
```

#### Types.typ - Exported data types
```iecst
TYPE
	HA_JSON_PairsToJSON_Internal_typ : 	STRUCT
		Depth : DINT;
		DepthArrayIdx : ARRAY[0..MAX_JSON_PARSE_DEPTH_IDX]OF DINT;
		Enabled : BOOL;
		j : DINT;
		i : DINT;
		Pair : HA_JSON_Parse_Pair_typ;
	END_STRUCT;
	HA_JSON_Parse_Internal_typ : 	STRUCT
		Depth : DINT;
		DepthArrayIdx : ARRAY[0..MAX_JSON_PARSE_DEPTH_IDX]OF DINT;
		DepthIDs : ARRAY[0..MAX_JSON_PARSE_DEPTH_IDX]OF STRING[MAX_JSON_PARSE_NAME_LEN];
		Marker : UDINT;
		InValueNonWhiteFound : BOOL;
		InValue : BOOL;
		InQuote : BOOL;
		QuoteIsDouble : BOOL;
		Send : BOOL;
		Idx : DINT;
		i : DINT;
		Enabled : BOOL;
		BufferLEN : UDINT;
		Pair : HA_JSON_Parse_Pair_typ;
	END_STRUCT;
	HA_JSON_Parse_Pair_typ : 	STRUCT
		Name : STRING[MAX_JSON_PARSE_NAME_LEN];
		Value : STRING[MAX_JSON_PARSE_VALUE_LEN];
	END_STRUCT;
END_TYPE
```

#### Constants.var - Exported constants
```iecst
VAR CONSTANT
	MAX_JSON_PARSE_DEPTH_IDX : DINT := 9;
	MAX_JSON_PARSE_PAIR_IDX : DINT := 10;
	MAX_JSON_PARSE_NAME_LEN : DINT := 40;
	MAX_JSON_PARSE_VALUE_LEN : DINT := 300;
END_VAR
```

#### HA_JSON_Parse.st
```iecst
(* FB parses a JSON string into a flat array of Name and Value Pairs, FOR LOOP COMPATIBLE *)FUNCTION_BLOCK HA_JSON_Parse

	IF Enable THEN
		IF NOT Internal.Enabled THEN
			brsmemset(ADR(Internal),0,SIZEOF(Internal));
			brsmemset(pPairs,0,(SIZEOF(Internal.Pair)*(MAX_JSON_PARSE_PAIR_IDX+1)));
			Internal.BufferLEN												:= brsstrlen(pBuffer);
			Internal.DepthArrayIdx[0]										:= -1;
			Internal.Enabled												:= TRUE;
		END_IF;
		IF Error OR Done THEN
			// Do Nothing, Enable must be toggled to parse again
		ELSE
			FOR Internal.i := 0 TO Internal.BufferLEN DO
				IF NOT Internal.InQuote THEN
					IF HA_Find_S(pBuffer+Internal.i,ADR('[')) >= 0 THEN													// New Array
						IF Internal.Depth <= MAX_JSON_PARSE_DEPTH_IDX THEN
							Internal.Depth 									:= Internal.Depth + 1;
							Internal.DepthIDs[Internal.Depth]				:= Internal.Pair.Name;
							IF Internal.DepthArrayIdx[Internal.Depth-1] >= 0 THEN
								Internal.Pair.Name							:= DINT_TO_STRING(Internal.DepthArrayIdx[Internal.Depth-1]);
								Internal.DepthArrayIdx[Internal.Depth-1] := Internal.DepthArrayIdx[Internal.Depth-1] + 1;
							END_IF;
							Internal.Pair.Value								:= '[';
							Internal.DepthIDs[Internal.Depth]				:= Internal.Pair.Name;
							Internal.DepthArrayIdx[Internal.Depth]			:= 0;
							Internal.Send									:= TRUE;
						ELSE
							Error											:= TRUE;
							EXIT;
						END_IF;
					ELSIF HA_Find_S(pBuffer+Internal.i,ADR('{')) >= 0 THEN 												// New Struct
						IF Internal.Depth <= MAX_JSON_PARSE_DEPTH_IDX THEN
							Internal.Depth 									:= Internal.Depth + 1;
							IF Internal.DepthArrayIdx[Internal.Depth-1] >= 0 THEN
								Internal.Pair.Name							:= DINT_TO_STRING(Internal.DepthArrayIdx[Internal.Depth-1]);
								Internal.DepthIDs[Internal.Depth]			:= Internal.Pair.Name;
								Internal.DepthArrayIdx[Internal.Depth-1] 	:= Internal.DepthArrayIdx[Internal.Depth-1] + 1;
								Internal.DepthArrayIdx[Internal.Depth]		:= -1;
								Internal.Pair.Value							:= '{';
								Internal.Send								:= TRUE;
							ELSE
								Internal.DepthIDs[Internal.Depth]			:= Internal.Pair.Name;
								Internal.DepthArrayIdx[Internal.Depth]		:= -1;
								Internal.Pair.Value							:= '{';
								Internal.Send								:= TRUE;
							END_IF;
						ELSE
							Error											:= TRUE;
							EXIT;
						END_IF;
					ELSIF HA_Find_S(pBuffer+Internal.i,ADR('"')) >= 0 THEN 												// New Double Quote
						Internal.InQuote									:= TRUE;
						Internal.QuoteIsDouble								:= TRUE;
						Internal.Marker										:= Internal.i+1;
						IF Internal.DepthArrayIdx[Internal.Depth] >= 0 THEN
							Internal.Pair.Name								:= DINT_TO_STRING(Internal.DepthArrayIdx[Internal.Depth]);
							Internal.DepthArrayIdx[Internal.Depth] 			:= Internal.DepthArrayIdx[Internal.Depth] + 1;
							Internal.InValue								:= TRUE;
						END_IF;
					ELSIF HA_Find_S(pBuffer+Internal.i,ADR('$'')) >= 0 THEN 											// New Single Quote
						Internal.InQuote									:= TRUE;
						Internal.QuoteIsDouble								:= FALSE;
						Internal.Marker										:= Internal.i+1;
						IF Internal.DepthArrayIdx[Internal.Depth] >= 0 THEN
							Internal.Pair.Name								:= DINT_TO_STRING(Internal.DepthArrayIdx[Internal.Depth]);
							Internal.DepthArrayIdx[Internal.Depth] 			:= Internal.DepthArrayIdx[Internal.Depth] + 1;
							Internal.InValue								:= TRUE;
						END_IF;
					ELSIF HA_Find_S(pBuffer+Internal.i,ADR(':')) >= 0 THEN
						// Value is next
						Internal.InValue									:= TRUE;
						Internal.Marker										:= Internal.i+1;
					ELSIF HA_Find_S(pBuffer+Internal.i,ADR(']')) >= 0 THEN
						IF Internal.InValue THEN
							Internal.InValue								:= FALSE;
							IF Internal.i <> 0 AND UDINT_TO_DINT(Internal.Marker) < Internal.i THEN
								IF (Internal.i - UDINT_TO_DINT(Internal.Marker)) < SIZEOF(Internal.Pair.Value) THEN
									brsmemcpy(ADR(Internal.Pair.Value),pBuffer+Internal.Marker,(Internal.i-Internal.Marker));
								ELSE
									brsmemcpy(ADR(Internal.Pair.Value),pBuffer+Internal.Marker,SIZEOF(Internal.Pair.Value)-1);
								END_IF;
								Internal.i 									:= Internal.i-1; 							// Go back one step to hit the bracket close again.
								Internal.Send								:= TRUE;
							ELSE
								Error										:= TRUE;
								EXIT;
							END_IF;
						ELSE
							Internal.DepthArrayIdx[Internal.Depth]			:= -1;
							Internal.Pair.Name								:= Internal.DepthIDs[Internal.Depth];
							Internal.DepthIDs[Internal.Depth]				:= '';
							Internal.Pair.Value								:= ']';
							Internal.Send									:= TRUE;
							IF Internal.Depth = 0 THEN
								Error										:= TRUE;
								EXIT;
							ELSE
								Internal.Depth								:= Internal.Depth - 1;
							END_IF;
						END_IF;
					ELSIF HA_Find_S(pBuffer+Internal.i,ADR('}')) >= 0 THEN
						IF Internal.InValue THEN
							Internal.InValue								:= FALSE;
							IF Internal.i <> 0 AND UDINT_TO_DINT(Internal.Marker) < Internal.i THEN
								IF (Internal.i - UDINT_TO_DINT(Internal.Marker)) < SIZEOF(Internal.Pair.Value) THEN
									brsmemcpy(ADR(Internal.Pair.Value),pBuffer+Internal.Marker,(Internal.i-Internal.Marker));
								ELSE
									brsmemcpy(ADR(Internal.Pair.Value),pBuffer+Internal.Marker,SIZEOF(Internal.Pair.Value)-1);
								END_IF;
								Internal.i 									:= Internal.i-1; 							// Go back one step to hit the bracket close again.
								Internal.Send								:= TRUE;
							ELSE
								Error										:= TRUE;
								EXIT;
							END_IF;
						ELSE
							Internal.DepthArrayIdx[Internal.Depth]			:= -1;
							Internal.Pair.Name								:= Internal.DepthIDs[Internal.Depth];
							Internal.DepthIDs[Internal.Depth]				:= '';
							Internal.Pair.Value								:= '}';
							Internal.Send									:= TRUE;
							IF Internal.Depth = 0 THEN
								Error										:= TRUE;
								EXIT;
							ELSE
								Internal.Depth								:= Internal.Depth - 1;
							END_IF;
						END_IF;
					ELSIF HA_Find_S(pBuffer+Internal.i,ADR(',')) >= 0 THEN
						IF Internal.InValue THEN
							Internal.InValue								:= FALSE;
							Internal.Send 									:= TRUE;
							IF Internal.i <> 0 AND UDINT_TO_DINT(Internal.Marker) < Internal.i THEN
								IF (Internal.i - UDINT_TO_DINT(Internal.Marker)) < SIZEOF(Internal.Pair.Value) THEN
									brsmemcpy(ADR(Internal.Pair.Value),pBuffer+Internal.Marker,(Internal.i-Internal.Marker));
								ELSE
									brsmemcpy(ADR(Internal.Pair.Value),pBuffer+Internal.Marker,SIZEOF(Internal.Pair.Value)-1);
								END_IF;
							ELSE
								Error										:= TRUE;
								EXIT;
							END_IF;
						END_IF;
					ELSIF HA_Find_S(pBuffer+Internal.i,ADR(' ')) >= 0 OR HA_Find_S(pBuffer+Internal.i,ADR('	')) >= 0 OR HA_Find_S(pBuffer+Internal.i,ADR('$r')) >= 0 OR HA_Find_S(pBuffer+Internal.i,ADR('$n')) >= 0 THEN //Whitespace
						IF NOT Internal.InValueNonWhiteFound THEN
							Internal.Marker									:= Internal.i+1;
						ELSIF Internal.InValue THEN
							Internal.InValue								:= FALSE;
							Internal.InValueNonWhiteFound					:= FALSE;
							IF Internal.i <> 0 AND UDINT_TO_DINT(Internal.Marker) < Internal.i THEN
								IF (Internal.i - UDINT_TO_DINT(Internal.Marker)) < SIZEOF(Internal.Pair.Value) THEN
									brsmemcpy(ADR(Internal.Pair.Value),pBuffer+Internal.Marker,(Internal.i-Internal.Marker));
								ELSE
									brsmemcpy(ADR(Internal.Pair.Value),pBuffer+Internal.Marker,SIZEOF(Internal.Pair.Value)-1);
								END_IF;
							ELSE
								Error										:= TRUE;
								EXIT;
							END_IF;
							Internal.Send 									:= TRUE;
						END_IF;
					ELSIF Internal.InValue OR Internal.DepthArrayIdx[Internal.Depth] >= 0 THEN
						Internal.InValue									:= TRUE;
						Internal.InValueNonWhiteFound						:= TRUE;
					END_IF;
				ELSIF Internal.QuoteIsDouble THEN 																		//Inside Double Quotes
					IF HA_Find_S(pBuffer+Internal.i,ADR('"')) >= 0 THEN
						IF Internal.InValue THEN
							Internal.InValue								:= FALSE;
							Internal.Send 									:= TRUE;
							IF Internal.i <> 0 AND UDINT_TO_DINT(Internal.Marker) < Internal.i THEN
								IF (Internal.i - UDINT_TO_DINT(Internal.Marker)) < SIZEOF(Internal.Pair.Value) THEN
									brsmemcpy(ADR(Internal.Pair.Value),ADR('"'),1);
									brsmemcpy(ADR(Internal.Pair.Value)+1,pBuffer+Internal.Marker,(Internal.i-Internal.Marker));
									brsmemcpy(ADR(Internal.Pair.Value)+1+(Internal.i-Internal.Marker),ADR('"'),1);
								ELSE
									brsmemcpy(ADR(Internal.Pair.Value),ADR('"'),1);
									brsmemcpy(ADR(Internal.Pair.Value)+1,pBuffer+Internal.Marker,SIZEOF(Internal.Pair.Value)-3);
									brsmemcpy(ADR(Internal.Pair.Value)+SIZEOF(Internal.Pair.Value)-1,ADR('"'),1);
								END_IF;
							ELSIF Internal.i <> 0 AND UDINT_TO_DINT(Internal.Marker) = Internal.i THEN
								brsmemcpy(ADR(Internal.Pair.Value),ADR('""'),2);
							ELSE
								Error										:= TRUE;
								EXIT;
							END_IF;
						ELSE
							IF Internal.i <> 0 AND UDINT_TO_DINT(Internal.Marker) < Internal.i THEN
								IF (Internal.i - UDINT_TO_DINT(Internal.Marker)) < SIZEOF(Internal.Pair.Name) THEN
									brsmemcpy(ADR(Internal.Pair.Name),pBuffer+Internal.Marker,(Internal.i-Internal.Marker));
								ELSE
									brsmemcpy(ADR(Internal.Pair.Name),pBuffer+Internal.Marker,SIZEOF(Internal.Pair.Name)-1);
								END_IF;
							ELSE
								Error										:= TRUE;
								EXIT;
							END_IF;
						END_IF;
						Internal.InQuote 									:= FALSE;
						Internal.QuoteIsDouble 								:= FALSE;
					END_IF;
				ELSE 																									//Inside Single Quotes
					IF HA_Find_S(pBuffer+Internal.i,ADR('$'')) >= 0 THEN
						IF Internal.InValue THEN
							Internal.InValue								:= FALSE;
							Internal.Send 									:= TRUE;
							IF Internal.i <> 0 AND UDINT_TO_DINT(Internal.Marker) < Internal.i THEN
								IF (Internal.i - UDINT_TO_DINT(Internal.Marker)) < SIZEOF(Internal.Pair.Value) THEN
									brsmemcpy(ADR(Internal.Pair.Value),ADR('$''),1);
									brsmemcpy(ADR(Internal.Pair.Value)+1,pBuffer+Internal.Marker,(Internal.i-Internal.Marker));
									brsmemcpy(ADR(Internal.Pair.Value)+1+(Internal.i-Internal.Marker),ADR('$''),1);
								ELSE
									brsmemcpy(ADR(Internal.Pair.Value),ADR('$''),1);
									brsmemcpy(ADR(Internal.Pair.Value)+1,pBuffer+Internal.Marker,SIZEOF(Internal.Pair.Value)-3);
									brsmemcpy(ADR(Internal.Pair.Value)+SIZEOF(Internal.Pair.Value)-1,ADR('$''),1);
								END_IF;
							ELSIF Internal.i <> 0 AND UDINT_TO_DINT(Internal.Marker) = Internal.i THEN
								brsmemcpy(ADR(Internal.Pair.Value),ADR('$'$''),2);
							ELSE
								Error										:= TRUE;
								EXIT;
							END_IF;
						ELSE
							IF Internal.i <> 0 AND UDINT_TO_DINT(Internal.Marker) < Internal.i THEN
								IF (Internal.i - UDINT_TO_DINT(Internal.Marker)) < SIZEOF(Internal.Pair.Name) THEN
									brsmemcpy(ADR(Internal.Pair.Name),pBuffer+Internal.Marker,(Internal.i-Internal.Marker));
								ELSE
									brsmemcpy(ADR(Internal.Pair.Name),pBuffer+Internal.Marker,SIZEOF(Internal.Pair.Name)-1);
								END_IF;
							ELSE
								Error										:= TRUE;
								EXIT;
							END_IF;
						END_IF;
						Internal.InQuote 									:= FALSE;
						Internal.QuoteIsDouble 								:= FALSE;
					END_IF;
				END_IF;
				IF Internal.Send THEN
					Internal.Send											:= FALSE;
					IF Internal.Idx >= 0 AND Internal.Idx <= MAX_JSON_PARSE_PAIR_IDX THEN
						brsmemcpy(pPairs+Internal.Idx*SIZEOF(Internal.Pair),ADR(Internal.Pair),SIZEOF(Internal.Pair));
						brsmemset(ADR(Internal.Pair),0,SIZEOF(Internal.Pair));
						Internal.InQuote									:= FALSE;
						Internal.InValue									:= FALSE;
						Internal.InValueNonWhiteFound						:= FALSE;
						Internal.Marker										:= 0;
						Internal.Idx										:= Internal.Idx + 1;
					ELSE
						Error												:= TRUE;
						EXIT;
					END_IF;
				END_IF;
			END_FOR;
			IF NOT Error THEN
				Done														:= TRUE;
			END_IF;
		END_IF;
	ELSE
		Done																:= FALSE;
		Error																:= FALSE;
		brsmemset(ADR(Internal),0,SIZEOF(Internal));
	END_IF;

END_FUNCTION_BLOCK
```

#### HA_JSON_PairsToJSON.st
```iecst
(* Takes Value Pairs and packs into a JSON String *)
FUNCTION_BLOCK HA_JSON_PairsToJSON
	IF Enable THEN
		IF NOT Internal.Enabled THEN
			brsmemset(ADR(Internal),0,SIZEOF(Internal));
			brsmemset(pBuffer,0,BufferSIZEOF);
			HA_brsstrcat(pBuffer,ADR('$r$n'),BufferSIZEOF);
			Internal.DepthArrayIdx[0]										:= -1;
			Internal.Enabled												:= TRUE;
		END_IF;
		IF Error OR Done THEN
			// Do Nothing, Enable must be toggled to parse again
		ELSE
			FOR Internal.i := 0 TO MAX_JSON_PARSE_PAIR_IDX DO
				brsmemcpy(ADR(Internal.Pair),pPairs+SIZEOF(Internal.Pair)*Internal.i,SIZEOF(Internal.Pair));
				IF Internal.Pair.Name = '' AND Internal.Pair.Value = '' THEN
					HA_brsstrcat(pBuffer,ADR('$r$n'),BufferSIZEOF);
					Done													:= TRUE;
					EXIT;
				ELSIF Internal.i = MAX_JSON_PARSE_PAIR_IDX AND Internal.Pair.Value <> '}' THEN
					Error													:= TRUE;
					EXIT;
				ELSE
					IF Internal.Pair.Value = '{' THEN
						IF Internal.Depth <= MAX_JSON_PARSE_DEPTH_IDX THEN
							Internal.Depth 									:= Internal.Depth + 1;
							Internal.DepthArrayIdx[Internal.Depth]			:= -1;
							IF Internal.DepthArrayIdx[Internal.Depth-1] >= 0 OR Internal.i = 0 THEN
								HA_brsstrcat(pBuffer,ADR('{'),BufferSIZEOF);
							ELSE
								HA_brsstrcat(pBuffer,ADR('"'),BufferSIZEOF);
								HA_brsstrcat(pBuffer,ADR(Internal.Pair.Name),BufferSIZEOF);
								HA_brsstrcat(pBuffer,ADR('": {'),BufferSIZEOF);
							END_IF;
							IF Internal.i <> MAX_JSON_PARSE_PAIR_IDX THEN
								brsmemcpy(ADR(Internal.Pair),pPairs+SIZEOF(Internal.Pair)*(Internal.i+1),SIZEOF(Internal.Pair));
								IF Internal.Pair.Value <> '}' THEN // Check next element to detect empty object condition
									HA_brsstrcat(pBuffer,ADR('$r$n'),BufferSIZEOF);
									FOR Internal.j := 0 TO (Internal.Depth-1)*2+1 DO
										HA_brsstrcat(pBuffer,ADR(' '),BufferSIZEOF);
									END_FOR;
								END_IF;
								brsmemcpy(ADR(Internal.Pair),pPairs+SIZEOF(Internal.Pair)*Internal.i,SIZEOF(Internal.Pair));
							END_IF;
						ELSE
							Error											:= TRUE;
							EXIT;
						END_IF;
					ELSIF Internal.Pair.Value = '}' THEN
						Internal.DepthArrayIdx[Internal.Depth]			:= -1;
						IF Internal.Depth = 0 THEN
							Error										:= TRUE;
							EXIT;
						ELSE
							Internal.Depth								:= Internal.Depth - 1;
						END_IF;
						HA_brsstrcat(pBuffer,ADR('}'),BufferSIZEOF);
						IF Internal.i <> MAX_JSON_PARSE_PAIR_IDX THEN
							brsmemcpy(ADR(Internal.Pair),pPairs+SIZEOF(Internal.Pair)*(Internal.i+1),SIZEOF(Internal.Pair));
							IF Internal.Pair.Value = '' AND Internal.Pair.Value = '' THEN

							ELSIF Internal.Pair.Value <> ']' AND Internal.Pair.Value <> '}' THEN
								HA_brsstrcat(pBuffer,ADR(','),BufferSIZEOF);
								HA_brsstrcat(pBuffer,ADR('$r$n'),BufferSIZEOF);
								FOR Internal.j := 0 TO (Internal.Depth-1)*2+1 DO
									HA_brsstrcat(pBuffer,ADR(' '),BufferSIZEOF);
								END_FOR;
							ELSE
								HA_brsstrcat(pBuffer,ADR('$r$n'),BufferSIZEOF);
								IF Internal.Depth >= 2 THEN
									FOR Internal.j := 0 TO (Internal.Depth-2)*2+1 DO
										HA_brsstrcat(pBuffer,ADR(' '),BufferSIZEOF);
									END_FOR;
								END_IF;
							END_IF;
							brsmemcpy(ADR(Internal.Pair),pPairs+SIZEOF(Internal.Pair)*Internal.i,SIZEOF(Internal.Pair));
						END_IF;
					ELSIF Internal.Pair.Value = '[' THEN
						IF Internal.Depth <= MAX_JSON_PARSE_DEPTH_IDX THEN
							Internal.Depth 									:= Internal.Depth + 1;
							Internal.DepthArrayIdx[Internal.Depth]			:= 0;
							IF Internal.DepthArrayIdx[Internal.Depth-1] >= 0 OR Internal.i = 0 THEN
								HA_brsstrcat(pBuffer,ADR('['),BufferSIZEOF);
							ELSE
								HA_brsstrcat(pBuffer,ADR('"'),BufferSIZEOF);
								HA_brsstrcat(pBuffer,ADR(Internal.Pair.Name),BufferSIZEOF);
								HA_brsstrcat(pBuffer,ADR('": ['),BufferSIZEOF);
							END_IF;
							IF Internal.i <> MAX_JSON_PARSE_PAIR_IDX THEN
								brsmemcpy(ADR(Internal.Pair),pPairs+SIZEOF(Internal.Pair)*(Internal.i+1),SIZEOF(Internal.Pair));
								IF Internal.Pair.Value = '[' OR Internal.Pair.Value = '{' THEN
									HA_brsstrcat(pBuffer,ADR('$r$n'),BufferSIZEOF);
									IF Internal.Depth >= 1 THEN
										FOR Internal.j := 0 TO (Internal.Depth-1)*2+1 DO
											HA_brsstrcat(pBuffer,ADR(' '),BufferSIZEOF);
										END_FOR;
									END_IF;
								END_IF;
								brsmemcpy(ADR(Internal.Pair),pPairs+SIZEOF(Internal.Pair)*Internal.i,SIZEOF(Internal.Pair));
							END_IF;
						ELSE
							Error											:= TRUE;
							EXIT;
						END_IF;
					ELSIF Internal.Pair.Value = ']' THEN
						Internal.DepthArrayIdx[Internal.Depth]			:= -1;
						IF Internal.Depth = 0 THEN
							Error										:= TRUE;
							EXIT;
						ELSE
							Internal.Depth								:= Internal.Depth - 1;
						END_IF;
						HA_brsstrcat(pBuffer,ADR(']'),BufferSIZEOF);
						IF Internal.i <> MAX_JSON_PARSE_PAIR_IDX THEN
							brsmemcpy(ADR(Internal.Pair),pPairs+SIZEOF(Internal.Pair)*(Internal.i+1),SIZEOF(Internal.Pair));
							IF Internal.Pair.Value = '' AND Internal.Pair.Value = '' THEN

							ELSIF Internal.Pair.Value <> ']' AND Internal.Pair.Value <> '}' THEN
								HA_brsstrcat(pBuffer,ADR(','),BufferSIZEOF);
								HA_brsstrcat(pBuffer,ADR('$r$n'),BufferSIZEOF);
								FOR Internal.j := 0 TO (Internal.Depth-1)*2+1 DO
									HA_brsstrcat(pBuffer,ADR(' '),BufferSIZEOF);
								END_FOR;
							ELSE
								HA_brsstrcat(pBuffer,ADR('$r$n'),BufferSIZEOF);
								IF Internal.Depth >= 2 THEN
									FOR Internal.j := 0 TO (Internal.Depth-2)*2+1 DO
										HA_brsstrcat(pBuffer,ADR(' '),BufferSIZEOF);
									END_FOR;
								END_IF;
							END_IF;
							brsmemcpy(ADR(Internal.Pair),pPairs+SIZEOF(Internal.Pair)*Internal.i,SIZEOF(Internal.Pair));
						END_IF;
					ELSE
						IF Internal.DepthArrayIdx[Internal.Depth] >= 0 THEN
							HA_brsstrcat(pBuffer,ADR(Internal.Pair.Value),BufferSIZEOF);
							IF Internal.i <> MAX_JSON_PARSE_PAIR_IDX THEN
								brsmemcpy(ADR(Internal.Pair),pPairs+SIZEOF(Internal.Pair)*(Internal.i+1),SIZEOF(Internal.Pair));
								IF Internal.Pair.Value <> ']' AND Internal.Pair.Value <> '}' THEN
									HA_brsstrcat(pBuffer,ADR(', '),BufferSIZEOF);
								END_IF;
								brsmemcpy(ADR(Internal.Pair),pPairs+SIZEOF(Internal.Pair)*Internal.i,SIZEOF(Internal.Pair));
							END_IF;
						ELSE
							HA_brsstrcat(pBuffer,ADR('"'),BufferSIZEOF);
							HA_brsstrcat(pBuffer,ADR(Internal.Pair.Name),BufferSIZEOF);
							HA_brsstrcat(pBuffer,ADR('": '),BufferSIZEOF);
							HA_brsstrcat(pBuffer,ADR(Internal.Pair.Value),BufferSIZEOF);
							IF Internal.i <> MAX_JSON_PARSE_PAIR_IDX THEN
								brsmemcpy(ADR(Internal.Pair),pPairs+SIZEOF(Internal.Pair)*(Internal.i+1),SIZEOF(Internal.Pair));
								IF Internal.Pair.Value <> ']' AND Internal.Pair.Value <> '}' THEN
									HA_brsstrcat(pBuffer,ADR(','),BufferSIZEOF);
									HA_brsstrcat(pBuffer,ADR('$r$n'),BufferSIZEOF);
									FOR Internal.j := 0 TO (Internal.Depth-1)*2+1 DO
										HA_brsstrcat(pBuffer,ADR(' '),BufferSIZEOF);
									END_FOR;
								ELSE
									HA_brsstrcat(pBuffer,ADR('$r$n'),BufferSIZEOF);
									IF Internal.Depth >= 2 THEN
										FOR Internal.j := 0 TO (Internal.Depth-2)*2+1 DO
											HA_brsstrcat(pBuffer,ADR(' '),BufferSIZEOF);
										END_FOR;
									END_IF;
								END_IF;
								brsmemcpy(ADR(Internal.Pair),pPairs+SIZEOF(Internal.Pair)*Internal.i,SIZEOF(Internal.Pair));
							END_IF;
						END_IF;
					END_IF;
				END_IF;
			END_FOR;
		END_IF;
	ELSE
		Done																:= FALSE;
		Error																:= FALSE;
		brsmemset(ADR(Internal),0,SIZEOF(Internal));
	END_IF;

END_FUNCTION_BLOCK
```

### Program Logical/modbusTCP/Master_HR (IEC) - modbusTCP master sample

#### ModMaster.var
```iecst
(*-----------------------------------------------------------------------------------------------------------------------------------------------------------------------------------------------------------------------------------------*)
(*Modbus master function block and configuration*)
VAR
	ModbusTcpMaster_HR : ARRAY[0..MAX_SKIDS_HR] OF MBmaster := [(0)];
	MasterConfig_HR : ARRAY[0..MAX_SKIDS_HR] OF modbus_master_cfg_typ := [(0)];
	reset_error : BOOL := FALSE;
END_VAR
(*IO sample arrays*)
VAR
	A_Out : ARRAY[0..255] OF UINT := [256(0)];
	UINT_In : ARRAY[0..50] OF UINT := [51(0)];
	REAL_In : ARRAY[0..50] OF REAL := [51(0.0)];
	D_Out : ARRAY[0..255] OF BOOL := [256(FALSE)];
	D_In : ARRAY[0..255] OF BOOL := [256(FALSE)];
END_VAR
(*MISC variables*)
VAR
	interface : STRING[20] := '';
	logger : ARRAY[0..LLN,0..MAX_SKIDS_HR] OF STRING[LLL] := [('')];
	StartStop : BOOL := FALSE;
	LREAL_Test : LREAL := 0.0;
	UDINT_Test : UDINT := 0;
	Test_REAL : ARRAY[0..3] OF REAL := [4(0)];
	Test_UDINT : UDINT := 0;
	Test_SWAPPED_UDINT : UDINT := 0;
	IdxReals : INT := 0;
	IdxUINTS : INT := 0;
	IdxSkids_HR : INT := 0;
	SkidString : STRING[80] := '';
	SkidNumberINT : STRING[80] := '';
	TestBool : BOOL := FALSE;
END_VAR
```
